REGION Network 54: Step[155] : Main P&P 1,2 Z-Axis Wait Pos
   RUNG wire#powerrail
      { S7_Templates := "SrcType := DInt" } EQ_Contact(in1 := "Unit1.Em4.ControlNodes".mainPnP.sequence.status.currentStep, in2 := #JOB_1_STEP_55)
      Contact( "Unit1.Em4.ControlNodes".mainPnP.sequence.status.seqActive )
      wire#w1
      Contact( #TRUE )
      wire#w2
      I_Contact( "Unit1.Em4.ControlNodes".cm.softCam.anodeMainPnP1AxisZ.upPos.inPos )
      wire#w3
      Coil( "Unit1.Em4.ControlNodes".mainPnP."step".action1[155] )
   END_RUNG
   RUNG wire#w2
      I_Contact( "Unit1.Em4.ControlNodes".cm.softCam.anodeMainPnP2AxisZ.upPos.inPos )
   END_RUNG wire#w3
   RUNG wire#w2
      Contact( "Unit1.Em4.ControlNodes".cm.softCam.anodeMainPnP1AxisZ.upPos.inPos )
      Contact( "Unit1.Em4.ControlNodes".cm.softCam.anodeMainPnP2AxisZ.upPos.inPos )
      Coil( "Unit1.Em4.ControlNodes".mainPnP."step".transition1[155] )
   END_RUNG
   RUNG wire#w1
      Contact( "Unit1.Em4.ControlNodes".mainPnP."step".transition1[155] )
      wire#w4
      { S7_Templates := "SrcType := DInt" } EQ_Contact(in1 := "Unit1.EmData".remainValue, in2 := 1)
      Contact( "Unit1.EmNodes".emRelations.em05.sequence.Spare1.selectJobStatus[1].completed )
      wire#w5
      Coil( "Unit1.Em4.ControlNodes".mainPnP."step".transition2[155] )
   END_RUNG
   RUNG wire#w4
      { S7_Templates := "SrcType := DInt" } EQ_Contact(in1 := "Unit1.EmData".remainValue, in2 := 0)
   END_RUNG wire#w5
   RUNG wire#w1
      Contact( "Unit1.Em4.ControlNodes".mainPnP."step".transition2[155] )
      { S7_Templates := "time_type := Time" } #statTonTime[155].TON(pt := #delayTime, et =>)
      Move(in := #JOB_1_STEP_80, out1 => "Unit1.Em4.ControlNodes".mainPnP.sequence.status.nextStep)
   END_RUNG
   // the same network as SCL:
   #_w1 := ("Unit1.Em4.ControlNodes".mainPnP.sequence.status.currentStep = #JOB_1_STEP_55) AND "Unit1.Em4.ControlNodes".mainPnP.sequence.status.seqActive;
   #_w2 := #_w1 AND #TRUE;
   "Unit1.Em4.ControlNodes".mainPnP."step".action1[155] := #_w2 AND (NOT "Unit1.Em4.ControlNodes".cm.softCam.anodeMainPnP1AxisZ.upPos.inPos OR NOT "Unit1.Em4.ControlNodes".cm.softCam.anodeMainPnP2AxisZ.upPos.inPos);
   "Unit1.Em4.ControlNodes".mainPnP."step".transition1[155] := #_w2 AND "Unit1.Em4.ControlNodes".cm.softCam.anodeMainPnP1AxisZ.upPos.inPos AND "Unit1.Em4.ControlNodes".cm.softCam.anodeMainPnP2AxisZ.upPos.inPos;
   "Unit1.Em4.ControlNodes".mainPnP."step".transition2[155] := #_w1 AND "Unit1.Em4.ControlNodes".mainPnP."step".transition1[155] AND ((("Unit1.EmData".remainValue = 1) AND "Unit1.EmNodes".emRelations.em05.sequence.Spare1.selectJobStatus[1].completed) OR ("Unit1.EmData".remainValue = 0));
   #statTonTime[155].TON(IN := #_w1 AND "Unit1.Em4.ControlNodes".mainPnP."step".transition2[155],
                         PT := #delayTime);
   IF #statTonTime[155].Q THEN
       "Unit1.Em4.ControlNodes".mainPnP.sequence.status.nextStep := #JOB_1_STEP_80;
   END_IF;
END_REGION

REGION Network 56: Step[180] : Main P&P 1,2 X-Axis Unload Pos
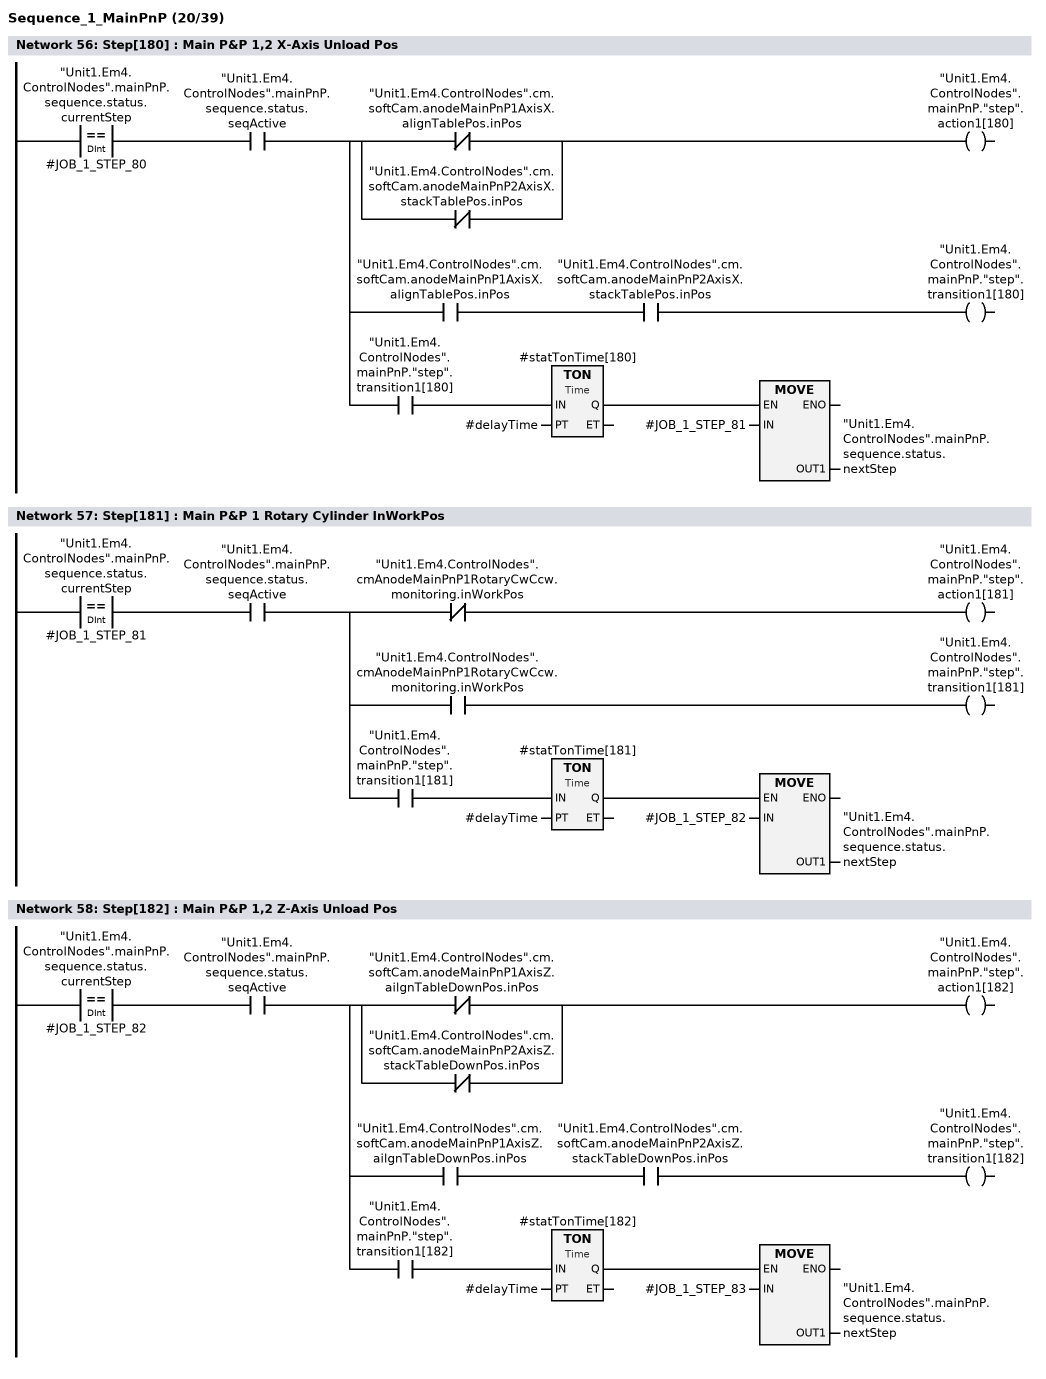
   RUNG wire#powerrail
      { S7_Templates := "SrcType := DInt" } EQ_Contact(in1 := "Unit1.Em4.ControlNodes".mainPnP.sequence.status.currentStep, in2 := #JOB_1_STEP_80)
      Contact( "Unit1.Em4.ControlNodes".mainPnP.sequence.status.seqActive )
      wire#w1
      I_Contact( "Unit1.Em4.ControlNodes".cm.softCam.anodeMainPnP1AxisX.alignTablePos.inPos )
      wire#w2
      Coil( "Unit1.Em4.ControlNodes".mainPnP."step".action1[180] )
   END_RUNG
   RUNG wire#w1
      I_Contact( "Unit1.Em4.ControlNodes".cm.softCam.anodeMainPnP2AxisX.stackTablePos.inPos )
   END_RUNG wire#w2
   RUNG wire#w1
      Contact( "Unit1.Em4.ControlNodes".cm.softCam.anodeMainPnP1AxisX.alignTablePos.inPos )
      Contact( "Unit1.Em4.ControlNodes".cm.softCam.anodeMainPnP2AxisX.stackTablePos.inPos )
      Coil( "Unit1.Em4.ControlNodes".mainPnP."step".transition1[180] )
   END_RUNG
   RUNG wire#w1
      Contact( "Unit1.Em4.ControlNodes".mainPnP."step".transition1[180] )
      { S7_Templates := "time_type := Time" } #statTonTime[180].TON(pt := #delayTime, et =>)
      Move(in := #JOB_1_STEP_81, out1 => "Unit1.Em4.ControlNodes".mainPnP.sequence.status.nextStep)
   END_RUNG
   // the same network as SCL:
   #_w1 := ("Unit1.Em4.ControlNodes".mainPnP.sequence.status.currentStep = #JOB_1_STEP_80) AND "Unit1.Em4.ControlNodes".mainPnP.sequence.status.seqActive;
   "Unit1.Em4.ControlNodes".mainPnP."step".action1[180] := #_w1 AND (NOT "Unit1.Em4.ControlNodes".cm.softCam.anodeMainPnP1AxisX.alignTablePos.inPos OR NOT "Unit1.Em4.ControlNodes".cm.softCam.anodeMainPnP2AxisX.stackTablePos.inPos);
   "Unit1.Em4.ControlNodes".mainPnP."step".transition1[180] := #_w1 AND "Unit1.Em4.ControlNodes".cm.softCam.anodeMainPnP1AxisX.alignTablePos.inPos AND "Unit1.Em4.ControlNodes".cm.softCam.anodeMainPnP2AxisX.stackTablePos.inPos;
   #statTonTime[180].TON(IN := #_w1 AND "Unit1.Em4.ControlNodes".mainPnP."step".transition1[180],
                         PT := #delayTime);
   IF #statTonTime[180].Q THEN
       "Unit1.Em4.ControlNodes".mainPnP.sequence.status.nextStep := #JOB_1_STEP_81;
   END_IF;
END_REGION

REGION Network 57: Step[181] : Main P&P 1 Rotary Cylinder InWorkPos
   RUNG wire#powerrail
      { S7_Templates := "SrcType := DInt" } EQ_Contact(in1 := "Unit1.Em4.ControlNodes".mainPnP.sequence.status.currentStep, in2 := #JOB_1_STEP_81)
      Contact( "Unit1.Em4.ControlNodes".mainPnP.sequence.status.seqActive )
      wire#w1
      I_Contact( "Unit1.Em4.ControlNodes".cmAnodeMainPnP1RotaryCwCcw.monitoring.inWorkPos )
      Coil( "Unit1.Em4.ControlNodes".mainPnP."step".action1[181] )
   END_RUNG
   RUNG wire#w1
      Contact( "Unit1.Em4.ControlNodes".cmAnodeMainPnP1RotaryCwCcw.monitoring.inWorkPos )
      Coil( "Unit1.Em4.ControlNodes".mainPnP."step".transition1[181] )
   END_RUNG
   RUNG wire#w1
      Contact( "Unit1.Em4.ControlNodes".mainPnP."step".transition1[181] )
      { S7_Templates := "time_type := Time" } #statTonTime[181].TON(pt := #delayTime, et =>)
      Move(in := #JOB_1_STEP_82, out1 => "Unit1.Em4.ControlNodes".mainPnP.sequence.status.nextStep)
   END_RUNG
   // the same network as SCL:
   #_w1 := ("Unit1.Em4.ControlNodes".mainPnP.sequence.status.currentStep = #JOB_1_STEP_81) AND "Unit1.Em4.ControlNodes".mainPnP.sequence.status.seqActive;
   "Unit1.Em4.ControlNodes".mainPnP."step".action1[181] := #_w1 AND NOT "Unit1.Em4.ControlNodes".cmAnodeMainPnP1RotaryCwCcw.monitoring.inWorkPos;
   "Unit1.Em4.ControlNodes".mainPnP."step".transition1[181] := #_w1 AND "Unit1.Em4.ControlNodes".cmAnodeMainPnP1RotaryCwCcw.monitoring.inWorkPos;
   #statTonTime[181].TON(IN := #_w1 AND "Unit1.Em4.ControlNodes".mainPnP."step".transition1[181],
                         PT := #delayTime);
   IF #statTonTime[181].Q THEN
       "Unit1.Em4.ControlNodes".mainPnP.sequence.status.nextStep := #JOB_1_STEP_82;
   END_IF;
END_REGION

REGION Network 58: Step[182] : Main P&P 1,2 Z-Axis Unload Pos
   RUNG wire#powerrail
      { S7_Templates := "SrcType := DInt" } EQ_Contact(in1 := "Unit1.Em4.ControlNodes".mainPnP.sequence.status.currentStep, in2 := #JOB_1_STEP_82)
      Contact( "Unit1.Em4.ControlNodes".mainPnP.sequence.status.seqActive )
      wire#w1
      I_Contact( "Unit1.Em4.ControlNodes".cm.softCam.anodeMainPnP1AxisZ.ailgnTableDownPos.inPos )
      wire#w2
      Coil( "Unit1.Em4.ControlNodes".mainPnP."step".action1[182] )
   END_RUNG
   RUNG wire#w1
      I_Contact( "Unit1.Em4.ControlNodes".cm.softCam.anodeMainPnP2AxisZ.stackTableDownPos.inPos )
   END_RUNG wire#w2
   RUNG wire#w1
      Contact( "Unit1.Em4.ControlNodes".cm.softCam.anodeMainPnP1AxisZ.ailgnTableDownPos.inPos )
      Contact( "Unit1.Em4.ControlNodes".cm.softCam.anodeMainPnP2AxisZ.stackTableDownPos.inPos )
      Coil( "Unit1.Em4.ControlNodes".mainPnP."step".transition1[182] )
   END_RUNG
   RUNG wire#w1
      Contact( "Unit1.Em4.ControlNodes".mainPnP."step".transition1[182] )
      { S7_Templates := "time_type := Time" } #statTonTime[182].TON(pt := #delayTime, et =>)
      Move(in := #JOB_1_STEP_83, out1 => "Unit1.Em4.ControlNodes".mainPnP.sequence.status.nextStep)
   END_RUNG
   // the same network as SCL:
   #_w1 := ("Unit1.Em4.ControlNodes".mainPnP.sequence.status.currentStep = #JOB_1_STEP_82) AND "Unit1.Em4.ControlNodes".mainPnP.sequence.status.seqActive;
   "Unit1.Em4.ControlNodes".mainPnP."step".action1[182] := #_w1 AND (NOT "Unit1.Em4.ControlNodes".cm.softCam.anodeMainPnP1AxisZ.ailgnTableDownPos.inPos OR NOT "Unit1.Em4.ControlNodes".cm.softCam.anodeMainPnP2AxisZ.stackTableDownPos.inPos);
   "Unit1.Em4.ControlNodes".mainPnP."step".transition1[182] := #_w1 AND "Unit1.Em4.ControlNodes".cm.softCam.anodeMainPnP1AxisZ.ailgnTableDownPos.inPos AND "Unit1.Em4.ControlNodes".cm.softCam.anodeMainPnP2AxisZ.stackTableDownPos.inPos;
   #statTonTime[182].TON(IN := #_w1 AND "Unit1.Em4.ControlNodes".mainPnP."step".transition1[182],
                         PT := #delayTime);
   IF #statTonTime[182].Q THEN
       "Unit1.Em4.ControlNodes".mainPnP.sequence.status.nextStep := #JOB_1_STEP_83;
   END_IF;
END_REGION

REGION Network 59: Step[183] : Main P&P → Align Table [Unloading Ready]
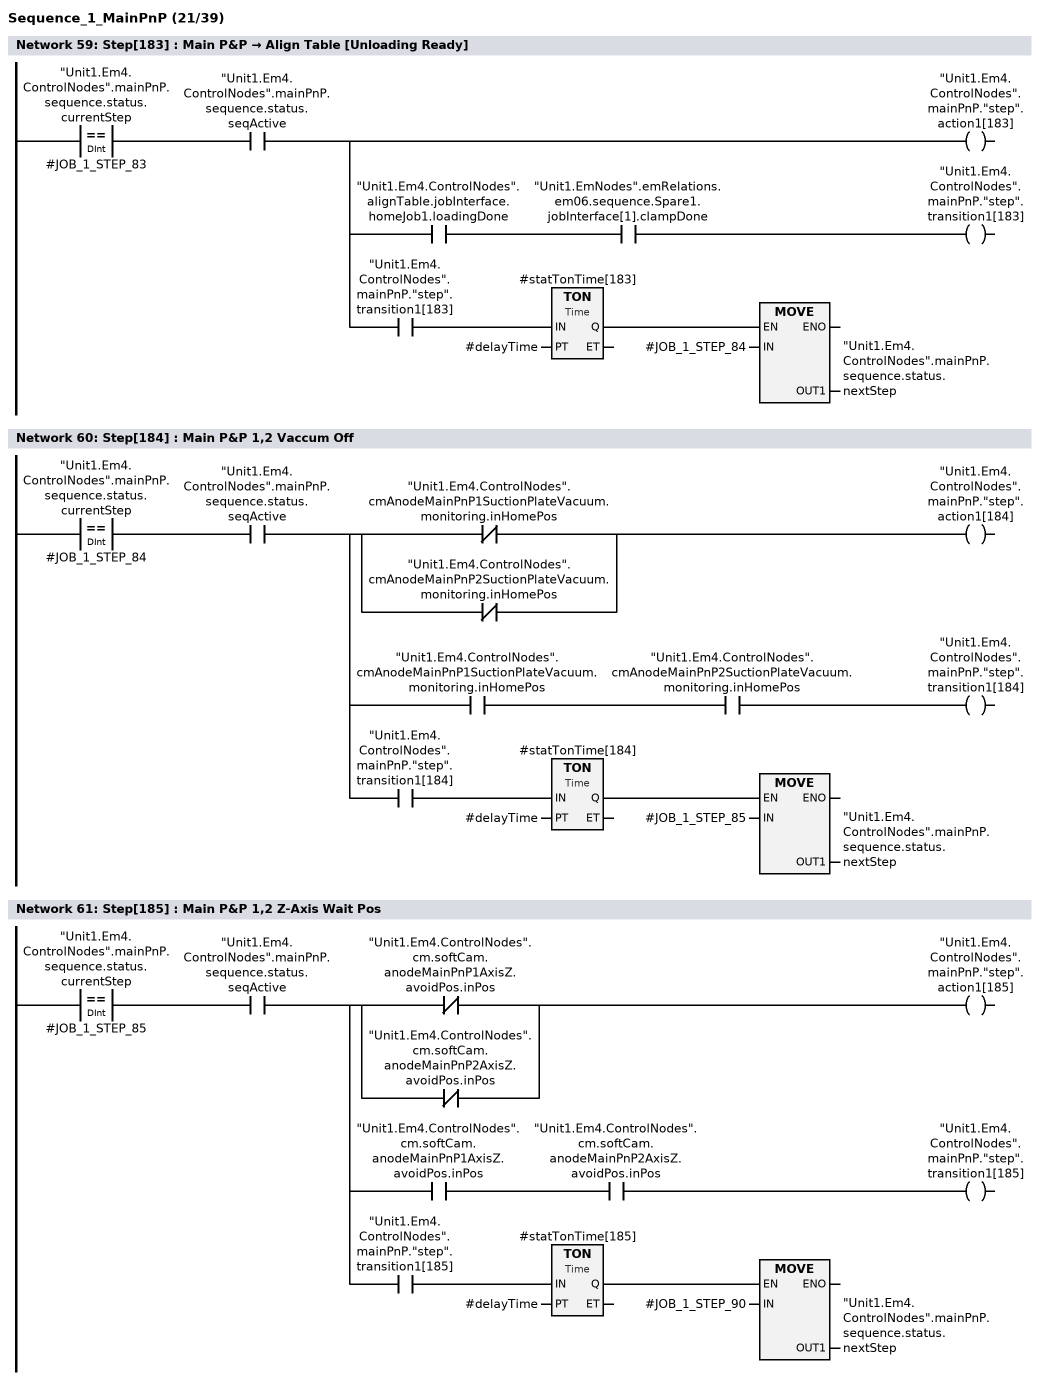
   RUNG wire#powerrail
      { S7_Templates := "SrcType := DInt" } EQ_Contact(in1 := "Unit1.Em4.ControlNodes".mainPnP.sequence.status.currentStep, in2 := #JOB_1_STEP_83)
      Contact( "Unit1.Em4.ControlNodes".mainPnP.sequence.status.seqActive )
      wire#w1
      Coil( "Unit1.Em4.ControlNodes".mainPnP."step".action1[183] )
   END_RUNG
   RUNG wire#w1
      Contact( "Unit1.Em4.ControlNodes".alignTable.jobInterface.homeJob1.loadingDone )
      Contact( "Unit1.EmNodes".emRelations.em06.sequence.Spare1.jobInterface[1].clampDone )
      Coil( "Unit1.Em4.ControlNodes".mainPnP."step".transition1[183] )
   END_RUNG
   RUNG wire#w1
      Contact( "Unit1.Em4.ControlNodes".mainPnP."step".transition1[183] )
      { S7_Templates := "time_type := Time" } #statTonTime[183].TON(pt := #delayTime, et =>)
      Move(in := #JOB_1_STEP_84, out1 => "Unit1.Em4.ControlNodes".mainPnP.sequence.status.nextStep)
   END_RUNG
   // the same network as SCL:
   "Unit1.Em4.ControlNodes".mainPnP."step".action1[183] := ("Unit1.Em4.ControlNodes".mainPnP.sequence.status.currentStep = #JOB_1_STEP_83) AND "Unit1.Em4.ControlNodes".mainPnP.sequence.status.seqActive;
   "Unit1.Em4.ControlNodes".mainPnP."step".transition1[183] := ("Unit1.Em4.ControlNodes".mainPnP.sequence.status.currentStep = #JOB_1_STEP_83) AND "Unit1.Em4.ControlNodes".mainPnP.sequence.status.seqActive AND "Unit1.Em4.ControlNodes".alignTable.jobInterface.homeJob1.loadingDone AND "Unit1.EmNodes".emRelations.em06.sequence.Spare1.jobInterface[1].clampDone;
   #statTonTime[183].TON(IN := ("Unit1.Em4.ControlNodes".mainPnP.sequence.status.currentStep = #JOB_1_STEP_83) AND "Unit1.Em4.ControlNodes".mainPnP.sequence.status.seqActive AND "Unit1.Em4.ControlNodes".mainPnP."step".transition1[183],
                         PT := #delayTime);
   IF #statTonTime[183].Q THEN
       "Unit1.Em4.ControlNodes".mainPnP.sequence.status.nextStep := #JOB_1_STEP_84;
   END_IF;
END_REGION

REGION Network 60: Step[184] : Main P&P 1,2 Vaccum Off
   RUNG wire#powerrail
      { S7_Templates := "SrcType := DInt" } EQ_Contact(in1 := "Unit1.Em4.ControlNodes".mainPnP.sequence.status.currentStep, in2 := #JOB_1_STEP_84)
      Contact( "Unit1.Em4.ControlNodes".mainPnP.sequence.status.seqActive )
      wire#w1
      I_Contact( "Unit1.Em4.ControlNodes".cmAnodeMainPnP1SuctionPlateVacuum.monitoring.inHomePos )
      wire#w2
      Coil( "Unit1.Em4.ControlNodes".mainPnP."step".action1[184] )
   END_RUNG
   RUNG wire#w1
      I_Contact( "Unit1.Em4.ControlNodes".cmAnodeMainPnP2SuctionPlateVacuum.monitoring.inHomePos )
   END_RUNG wire#w2
   RUNG wire#w1
      Contact( "Unit1.Em4.ControlNodes".cmAnodeMainPnP1SuctionPlateVacuum.monitoring.inHomePos )
      Contact( "Unit1.Em4.ControlNodes".cmAnodeMainPnP2SuctionPlateVacuum.monitoring.inHomePos )
      Coil( "Unit1.Em4.ControlNodes".mainPnP."step".transition1[184] )
   END_RUNG
   RUNG wire#w1
      Contact( "Unit1.Em4.ControlNodes".mainPnP."step".transition1[184] )
      { S7_Templates := "time_type := Time" } #statTonTime[184].TON(pt := #delayTime, et =>)
      Move(in := #JOB_1_STEP_85, out1 => "Unit1.Em4.ControlNodes".mainPnP.sequence.status.nextStep)
   END_RUNG
   // the same network as SCL:
   #_w1 := ("Unit1.Em4.ControlNodes".mainPnP.sequence.status.currentStep = #JOB_1_STEP_84) AND "Unit1.Em4.ControlNodes".mainPnP.sequence.status.seqActive;
   "Unit1.Em4.ControlNodes".mainPnP."step".action1[184] := #_w1 AND (NOT "Unit1.Em4.ControlNodes".cmAnodeMainPnP1SuctionPlateVacuum.monitoring.inHomePos OR NOT "Unit1.Em4.ControlNodes".cmAnodeMainPnP2SuctionPlateVacuum.monitoring.inHomePos);
   "Unit1.Em4.ControlNodes".mainPnP."step".transition1[184] := #_w1 AND "Unit1.Em4.ControlNodes".cmAnodeMainPnP1SuctionPlateVacuum.monitoring.inHomePos AND "Unit1.Em4.ControlNodes".cmAnodeMainPnP2SuctionPlateVacuum.monitoring.inHomePos;
   #statTonTime[184].TON(IN := #_w1 AND "Unit1.Em4.ControlNodes".mainPnP."step".transition1[184],
                         PT := #delayTime);
   IF #statTonTime[184].Q THEN
       "Unit1.Em4.ControlNodes".mainPnP.sequence.status.nextStep := #JOB_1_STEP_85;
   END_IF;
END_REGION

REGION Network 61: Step[185] : Main P&P 1,2 Z-Axis Wait Pos
   RUNG wire#powerrail
      { S7_Templates := "SrcType := DInt" } EQ_Contact(in1 := "Unit1.Em4.ControlNodes".mainPnP.sequence.status.currentStep, in2 := #JOB_1_STEP_85)
      Contact( "Unit1.Em4.ControlNodes".mainPnP.sequence.status.seqActive )
      wire#w1
      I_Contact( "Unit1.Em4.ControlNodes".cm.softCam.anodeMainPnP1AxisZ.avoidPos.inPos )
      wire#w2
      Coil( "Unit1.Em4.ControlNodes".mainPnP."step".action1[185] )
   END_RUNG
   RUNG wire#w1
      I_Contact( "Unit1.Em4.ControlNodes".cm.softCam.anodeMainPnP2AxisZ.avoidPos.inPos )
   END_RUNG wire#w2
   RUNG wire#w1
      Contact( "Unit1.Em4.ControlNodes".cm.softCam.anodeMainPnP1AxisZ.avoidPos.inPos )
      Contact( "Unit1.Em4.ControlNodes".cm.softCam.anodeMainPnP2AxisZ.avoidPos.inPos )
      Coil( "Unit1.Em4.ControlNodes".mainPnP."step".transition1[185] )
   END_RUNG
   RUNG wire#w1
      Contact( "Unit1.Em4.ControlNodes".mainPnP."step".transition1[185] )
      { S7_Templates := "time_type := Time" } #statTonTime[185].TON(pt := #delayTime, et =>)
      Move(in := #JOB_1_STEP_90, out1 => "Unit1.Em4.ControlNodes".mainPnP.sequence.status.nextStep)
   END_RUNG
   // the same network as SCL:
   #_w1 := ("Unit1.Em4.ControlNodes".mainPnP.sequence.status.currentStep = #JOB_1_STEP_85) AND "Unit1.Em4.ControlNodes".mainPnP.sequence.status.seqActive;
   "Unit1.Em4.ControlNodes".mainPnP."step".action1[185] := #_w1 AND (NOT "Unit1.Em4.ControlNodes".cm.softCam.anodeMainPnP1AxisZ.avoidPos.inPos OR NOT "Unit1.Em4.ControlNodes".cm.softCam.anodeMainPnP2AxisZ.avoidPos.inPos);
   "Unit1.Em4.ControlNodes".mainPnP."step".transition1[185] := #_w1 AND "Unit1.Em4.ControlNodes".cm.softCam.anodeMainPnP1AxisZ.avoidPos.inPos AND "Unit1.Em4.ControlNodes".cm.softCam.anodeMainPnP2AxisZ.avoidPos.inPos;
   #statTonTime[185].TON(IN := #_w1 AND "Unit1.Em4.ControlNodes".mainPnP."step".transition1[185],
                         PT := #delayTime);
   IF #statTonTime[185].Q THEN
       "Unit1.Em4.ControlNodes".mainPnP.sequence.status.nextStep := #JOB_1_STEP_90;
   END_IF;
END_REGION

REGION Network 62: Step[190] : JOB[1] Step End
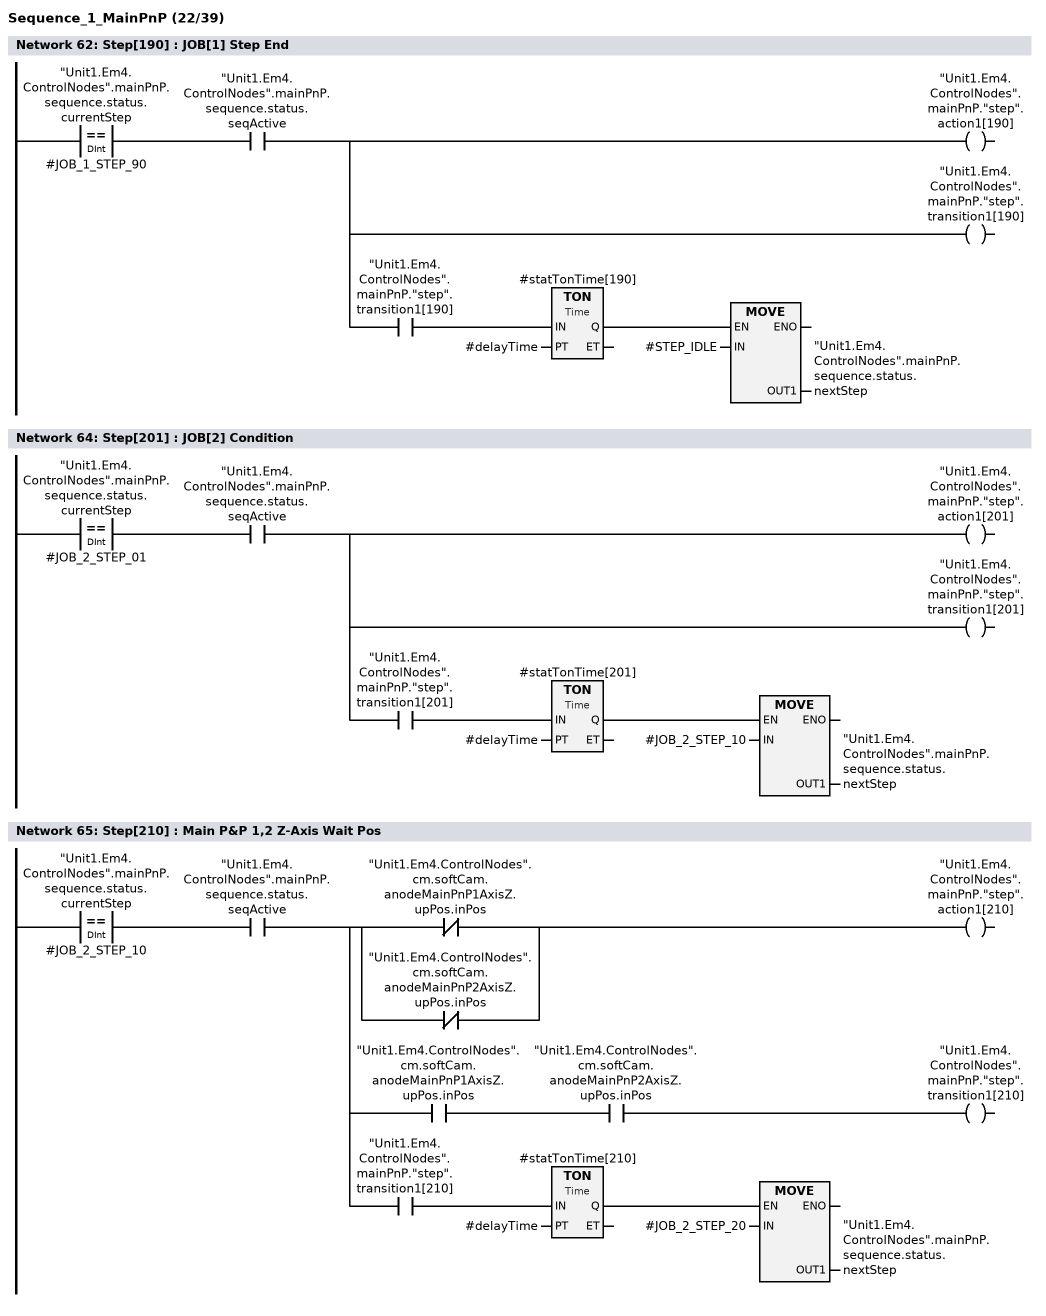
   RUNG wire#powerrail
      { S7_Templates := "SrcType := DInt" } EQ_Contact(in1 := "Unit1.Em4.ControlNodes".mainPnP.sequence.status.currentStep, in2 := #JOB_1_STEP_90)
      Contact( "Unit1.Em4.ControlNodes".mainPnP.sequence.status.seqActive )
      wire#w1
      Coil( "Unit1.Em4.ControlNodes".mainPnP."step".action1[190] )
   END_RUNG
   RUNG wire#w1
      Coil( "Unit1.Em4.ControlNodes".mainPnP."step".transition1[190] )
   END_RUNG
   RUNG wire#w1
      Contact( "Unit1.Em4.ControlNodes".mainPnP."step".transition1[190] )
      { S7_Templates := "time_type := Time" } #statTonTime[190].TON(pt := #delayTime, et =>)
      Move(in := #STEP_IDLE, out1 => "Unit1.Em4.ControlNodes".mainPnP.sequence.status.nextStep)
   END_RUNG
   // the same network as SCL:
   "Unit1.Em4.ControlNodes".mainPnP."step".action1[190] := ("Unit1.Em4.ControlNodes".mainPnP.sequence.status.currentStep = #JOB_1_STEP_90) AND "Unit1.Em4.ControlNodes".mainPnP.sequence.status.seqActive;
   "Unit1.Em4.ControlNodes".mainPnP."step".transition1[190] := ("Unit1.Em4.ControlNodes".mainPnP.sequence.status.currentStep = #JOB_1_STEP_90) AND "Unit1.Em4.ControlNodes".mainPnP.sequence.status.seqActive;
   #statTonTime[190].TON(IN := ("Unit1.Em4.ControlNodes".mainPnP.sequence.status.currentStep = #JOB_1_STEP_90) AND "Unit1.Em4.ControlNodes".mainPnP.sequence.status.seqActive AND "Unit1.Em4.ControlNodes".mainPnP."step".transition1[190],
                         PT := #delayTime);
   IF #statTonTime[190].Q THEN
       "Unit1.Em4.ControlNodes".mainPnP.sequence.status.nextStep := #STEP_IDLE;
   END_IF;
END_REGION

REGION Network 63: *************** JOB[2] Loading ************************
END_REGION

REGION Network 64: Step[201] : JOB[2] Condition
   RUNG wire#powerrail
      { S7_Templates := "SrcType := DInt" } EQ_Contact(in1 := "Unit1.Em4.ControlNodes".mainPnP.sequence.status.currentStep, in2 := #JOB_2_STEP_01)
      Contact( "Unit1.Em4.ControlNodes".mainPnP.sequence.status.seqActive )
      wire#w1
      Coil( "Unit1.Em4.ControlNodes".mainPnP."step".action1[201] )
   END_RUNG
   RUNG wire#w1
      Coil( "Unit1.Em4.ControlNodes".mainPnP."step".transition1[201] )
   END_RUNG
   RUNG wire#w1
      Contact( "Unit1.Em4.ControlNodes".mainPnP."step".transition1[201] )
      { S7_Templates := "time_type := Time" } #statTonTime[201].TON(pt := #delayTime, et =>)
      Move(in := #JOB_2_STEP_10, out1 => "Unit1.Em4.ControlNodes".mainPnP.sequence.status.nextStep)
   END_RUNG
   // the same network as SCL:
   "Unit1.Em4.ControlNodes".mainPnP."step".action1[201] := ("Unit1.Em4.ControlNodes".mainPnP.sequence.status.currentStep = #JOB_2_STEP_01) AND "Unit1.Em4.ControlNodes".mainPnP.sequence.status.seqActive;
   "Unit1.Em4.ControlNodes".mainPnP."step".transition1[201] := ("Unit1.Em4.ControlNodes".mainPnP.sequence.status.currentStep = #JOB_2_STEP_01) AND "Unit1.Em4.ControlNodes".mainPnP.sequence.status.seqActive;
   #statTonTime[201].TON(IN := ("Unit1.Em4.ControlNodes".mainPnP.sequence.status.currentStep = #JOB_2_STEP_01) AND "Unit1.Em4.ControlNodes".mainPnP.sequence.status.seqActive AND "Unit1.Em4.ControlNodes".mainPnP."step".transition1[201],
                         PT := #delayTime);
   IF #statTonTime[201].Q THEN
       "Unit1.Em4.ControlNodes".mainPnP.sequence.status.nextStep := #JOB_2_STEP_10;
   END_IF;
END_REGION

REGION Network 65: Step[210] : Main P&P 1,2 Z-Axis Wait Pos
   RUNG wire#powerrail
      { S7_Templates := "SrcType := DInt" } EQ_Contact(in1 := "Unit1.Em4.ControlNodes".mainPnP.sequence.status.currentStep, in2 := #JOB_2_STEP_10)
      Contact( "Unit1.Em4.ControlNodes".mainPnP.sequence.status.seqActive )
      wire#w1
      I_Contact( "Unit1.Em4.ControlNodes".cm.softCam.anodeMainPnP1AxisZ.upPos.inPos )
      wire#w2
      Coil( "Unit1.Em4.ControlNodes".mainPnP."step".action1[210] )
   END_RUNG
   RUNG wire#w1
      I_Contact( "Unit1.Em4.ControlNodes".cm.softCam.anodeMainPnP2AxisZ.upPos.inPos )
   END_RUNG wire#w2
   RUNG wire#w1
      Contact( "Unit1.Em4.ControlNodes".cm.softCam.anodeMainPnP1AxisZ.upPos.inPos )
      Contact( "Unit1.Em4.ControlNodes".cm.softCam.anodeMainPnP2AxisZ.upPos.inPos )
      Coil( "Unit1.Em4.ControlNodes".mainPnP."step".transition1[210] )
   END_RUNG
   RUNG wire#w1
      Contact( "Unit1.Em4.ControlNodes".mainPnP."step".transition1[210] )
      { S7_Templates := "time_type := Time" } #statTonTime[210].TON(pt := #delayTime, et =>)
      Move(in := #JOB_2_STEP_20, out1 => "Unit1.Em4.ControlNodes".mainPnP.sequence.status.nextStep)
   END_RUNG
   // the same network as SCL:
   #_w1 := ("Unit1.Em4.ControlNodes".mainPnP.sequence.status.currentStep = #JOB_2_STEP_10) AND "Unit1.Em4.ControlNodes".mainPnP.sequence.status.seqActive;
   "Unit1.Em4.ControlNodes".mainPnP."step".action1[210] := #_w1 AND (NOT "Unit1.Em4.ControlNodes".cm.softCam.anodeMainPnP1AxisZ.upPos.inPos OR NOT "Unit1.Em4.ControlNodes".cm.softCam.anodeMainPnP2AxisZ.upPos.inPos);
   "Unit1.Em4.ControlNodes".mainPnP."step".transition1[210] := #_w1 AND "Unit1.Em4.ControlNodes".cm.softCam.anodeMainPnP1AxisZ.upPos.inPos AND "Unit1.Em4.ControlNodes".cm.softCam.anodeMainPnP2AxisZ.upPos.inPos;
   #statTonTime[210].TON(IN := #_w1 AND "Unit1.Em4.ControlNodes".mainPnP."step".transition1[210],
                         PT := #delayTime);
   IF #statTonTime[210].Q THEN
       "Unit1.Em4.ControlNodes".mainPnP.sequence.status.nextStep := #JOB_2_STEP_20;
   END_IF;
END_REGION

REGION Network 66: Step[220] : Main P&P 1,2 X-Axis Load Pos
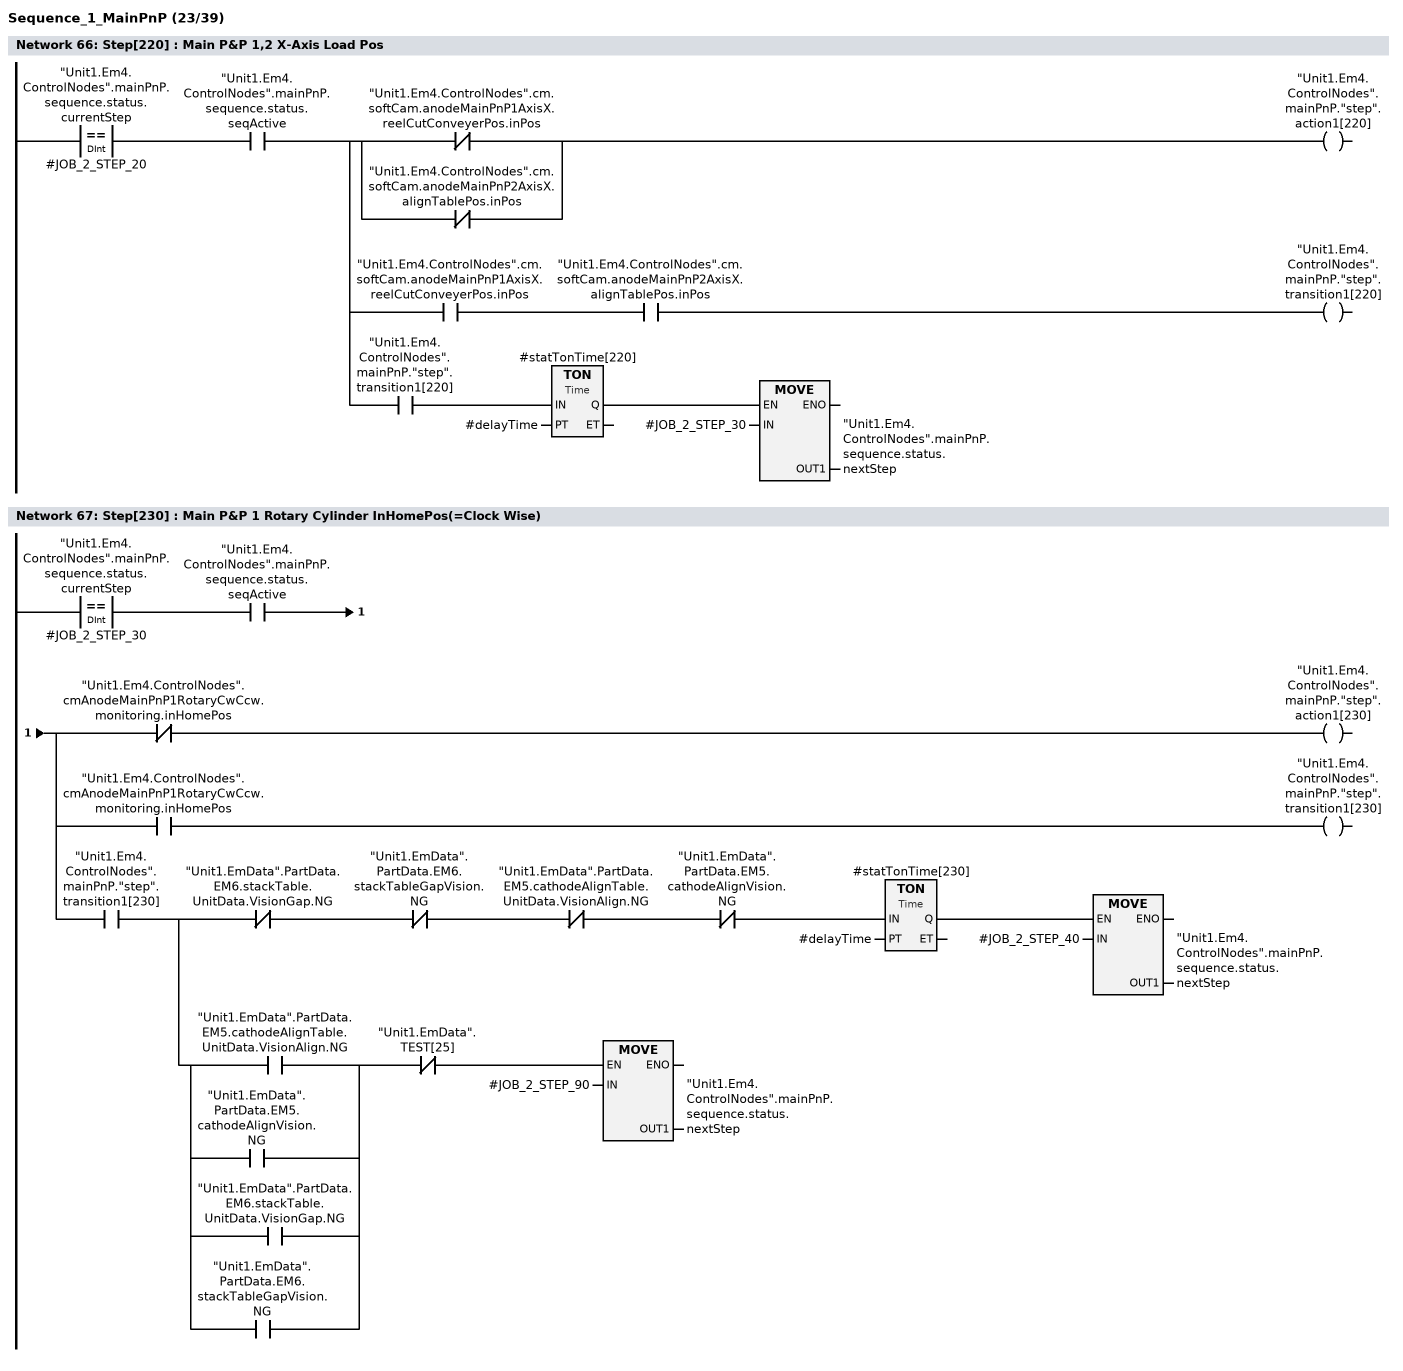
   RUNG wire#powerrail
      { S7_Templates := "SrcType := DInt" } EQ_Contact(in1 := "Unit1.Em4.ControlNodes".mainPnP.sequence.status.currentStep, in2 := #JOB_2_STEP_20)
      Contact( "Unit1.Em4.ControlNodes".mainPnP.sequence.status.seqActive )
      wire#w1
      I_Contact( "Unit1.Em4.ControlNodes".cm.softCam.anodeMainPnP1AxisX.reelCutConveyerPos.inPos )
      wire#w2
      Coil( "Unit1.Em4.ControlNodes".mainPnP."step".action1[220] )
   END_RUNG
   RUNG wire#w1
      I_Contact( "Unit1.Em4.ControlNodes".cm.softCam.anodeMainPnP2AxisX.alignTablePos.inPos )
   END_RUNG wire#w2
   RUNG wire#w1
      Contact( "Unit1.Em4.ControlNodes".cm.softCam.anodeMainPnP1AxisX.reelCutConveyerPos.inPos )
      Contact( "Unit1.Em4.ControlNodes".cm.softCam.anodeMainPnP2AxisX.alignTablePos.inPos )
      Coil( "Unit1.Em4.ControlNodes".mainPnP."step".transition1[220] )
   END_RUNG
   RUNG wire#w1
      Contact( "Unit1.Em4.ControlNodes".mainPnP."step".transition1[220] )
      { S7_Templates := "time_type := Time" } #statTonTime[220].TON(pt := #delayTime, et =>)
      Move(in := #JOB_2_STEP_30, out1 => "Unit1.Em4.ControlNodes".mainPnP.sequence.status.nextStep)
   END_RUNG
   // the same network as SCL:
   #_w1 := ("Unit1.Em4.ControlNodes".mainPnP.sequence.status.currentStep = #JOB_2_STEP_20) AND "Unit1.Em4.ControlNodes".mainPnP.sequence.status.seqActive;
   "Unit1.Em4.ControlNodes".mainPnP."step".action1[220] := #_w1 AND (NOT "Unit1.Em4.ControlNodes".cm.softCam.anodeMainPnP1AxisX.reelCutConveyerPos.inPos OR NOT "Unit1.Em4.ControlNodes".cm.softCam.anodeMainPnP2AxisX.alignTablePos.inPos);
   "Unit1.Em4.ControlNodes".mainPnP."step".transition1[220] := #_w1 AND "Unit1.Em4.ControlNodes".cm.softCam.anodeMainPnP1AxisX.reelCutConveyerPos.inPos AND "Unit1.Em4.ControlNodes".cm.softCam.anodeMainPnP2AxisX.alignTablePos.inPos;
   #statTonTime[220].TON(IN := #_w1 AND "Unit1.Em4.ControlNodes".mainPnP."step".transition1[220],
                         PT := #delayTime);
   IF #statTonTime[220].Q THEN
       "Unit1.Em4.ControlNodes".mainPnP.sequence.status.nextStep := #JOB_2_STEP_30;
   END_IF;
END_REGION

REGION Network 67: Step[230] : Main P&P 1 Rotary Cylinder InHomePos(=Clock Wise)
   RUNG wire#powerrail
      { S7_Templates := "SrcType := DInt" } EQ_Contact(in1 := "Unit1.Em4.ControlNodes".mainPnP.sequence.status.currentStep, in2 := #JOB_2_STEP_30)
      Contact( "Unit1.Em4.ControlNodes".mainPnP.sequence.status.seqActive )
      wire#w1
      I_Contact( "Unit1.Em4.ControlNodes".cmAnodeMainPnP1RotaryCwCcw.monitoring.inHomePos )
      Coil( "Unit1.Em4.ControlNodes".mainPnP."step".action1[230] )
   END_RUNG
   RUNG wire#w1
      Contact( "Unit1.Em4.ControlNodes".cmAnodeMainPnP1RotaryCwCcw.monitoring.inHomePos )
      Coil( "Unit1.Em4.ControlNodes".mainPnP."step".transition1[230] )
   END_RUNG
   RUNG wire#w1
      Contact( "Unit1.Em4.ControlNodes".mainPnP."step".transition1[230] )
      wire#w2
      I_Contact( "Unit1.EmData".PartData.EM6.stackTable.UnitData.VisionGap.NG )
      I_Contact( "Unit1.EmData".PartData.EM6.stackTableGapVision.NG )
      I_Contact( "Unit1.EmData".PartData.EM5.cathodeAlignTable.UnitData.VisionAlign.NG )
      I_Contact( "Unit1.EmData".PartData.EM5.cathodeAlignVision.NG )
      { S7_Templates := "time_type := Time" } #statTonTime[230].TON(pt := #delayTime, et =>)
      Move(in := #JOB_2_STEP_40, out1 => "Unit1.Em4.ControlNodes".mainPnP.sequence.status.nextStep)
   END_RUNG
   RUNG wire#w2
      Contact( "Unit1.EmData".PartData.EM5.cathodeAlignTable.UnitData.VisionAlign.NG )
      wire#w3
      I_Contact( "Unit1.EmData".TEST[25] )
      Move(in := #JOB_2_STEP_90, out1 => "Unit1.Em4.ControlNodes".mainPnP.sequence.status.nextStep)
   END_RUNG
   RUNG wire#w2
      Contact( "Unit1.EmData".PartData.EM5.cathodeAlignVision.NG )
   END_RUNG wire#w3
   RUNG wire#w2
      Contact( "Unit1.EmData".PartData.EM6.stackTable.UnitData.VisionGap.NG )
   END_RUNG wire#w3
   RUNG wire#w2
      Contact( "Unit1.EmData".PartData.EM6.stackTableGapVision.NG )
   END_RUNG wire#w3
   // the same network as SCL:
   #_w1 := ("Unit1.Em4.ControlNodes".mainPnP.sequence.status.currentStep = #JOB_2_STEP_30) AND "Unit1.Em4.ControlNodes".mainPnP.sequence.status.seqActive;
   "Unit1.Em4.ControlNodes".mainPnP."step".action1[230] := #_w1 AND NOT "Unit1.Em4.ControlNodes".cmAnodeMainPnP1RotaryCwCcw.monitoring.inHomePos;
   "Unit1.Em4.ControlNodes".mainPnP."step".transition1[230] := #_w1 AND "Unit1.Em4.ControlNodes".cmAnodeMainPnP1RotaryCwCcw.monitoring.inHomePos;
   #_w2 := #_w1 AND "Unit1.Em4.ControlNodes".mainPnP."step".transition1[230];
   #statTonTime[230].TON(IN := #_w2 AND NOT "Unit1.EmData".PartData.EM6.stackTable.UnitData.VisionGap.NG AND NOT "Unit1.EmData".PartData.EM6.stackTableGapVision.NG AND NOT "Unit1.EmData".PartData.EM5.cathodeAlignTable.UnitData.VisionAlign.NG AND NOT "Unit1.EmData".PartData.EM5.cathodeAlignVision.NG,
                         PT := #delayTime);
   IF #statTonTime[230].Q THEN
       "Unit1.Em4.ControlNodes".mainPnP.sequence.status.nextStep := #JOB_2_STEP_40;
   END_IF;
   IF #_w2 AND ("Unit1.EmData".PartData.EM5.cathodeAlignTable.UnitData.VisionAlign.NG OR "Unit1.EmData".PartData.EM5.cathodeAlignVision.NG OR "Unit1.EmData".PartData.EM6.stackTable.UnitData.VisionGap.NG OR "Unit1.EmData".PartData.EM6.stackTableGapVision.NG) AND NOT "Unit1.EmData".TEST[25] THEN
       "Unit1.Em4.ControlNodes".mainPnP.sequence.status.nextStep := #JOB_2_STEP_90;
   END_IF;
END_REGION

REGION Network 68: Step[240] : Main P&P 1.2 Z-Axis Load Pos
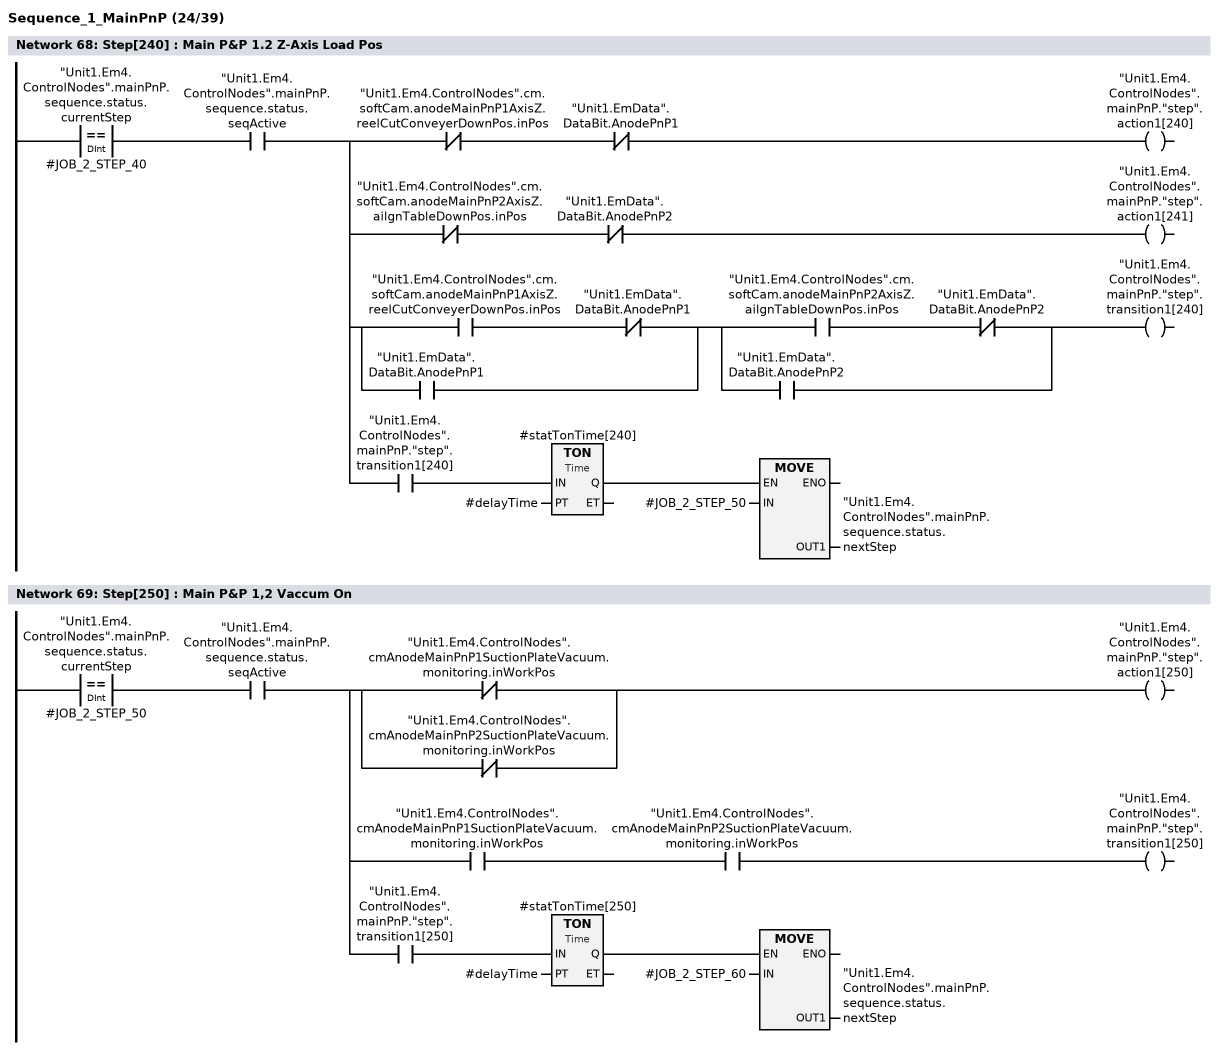
   RUNG wire#powerrail
      { S7_Templates := "SrcType := DInt" } EQ_Contact(in1 := "Unit1.Em4.ControlNodes".mainPnP.sequence.status.currentStep, in2 := #JOB_2_STEP_40)
      Contact( "Unit1.Em4.ControlNodes".mainPnP.sequence.status.seqActive )
      wire#w1
      I_Contact( "Unit1.Em4.ControlNodes".cm.softCam.anodeMainPnP1AxisZ.reelCutConveyerDownPos.inPos )
      I_Contact( "Unit1.EmData".DataBit.AnodePnP1 )
      Coil( "Unit1.Em4.ControlNodes".mainPnP."step".action1[240] )
   END_RUNG
   RUNG wire#w1
      I_Contact( "Unit1.Em4.ControlNodes".cm.softCam.anodeMainPnP2AxisZ.ailgnTableDownPos.inPos )
      I_Contact( "Unit1.EmData".DataBit.AnodePnP2 )
      Coil( "Unit1.Em4.ControlNodes".mainPnP."step".action1[241] )
   END_RUNG
   RUNG wire#w1
      Contact( "Unit1.Em4.ControlNodes".cm.softCam.anodeMainPnP1AxisZ.reelCutConveyerDownPos.inPos )
      I_Contact( "Unit1.EmData".DataBit.AnodePnP1 )
      wire#w2
      Contact( "Unit1.Em4.ControlNodes".cm.softCam.anodeMainPnP2AxisZ.ailgnTableDownPos.inPos )
      I_Contact( "Unit1.EmData".DataBit.AnodePnP2 )
      wire#w3
      Coil( "Unit1.Em4.ControlNodes".mainPnP."step".transition1[240] )
   END_RUNG
   RUNG wire#w1
      Contact( "Unit1.EmData".DataBit.AnodePnP1 )
   END_RUNG wire#w2
   RUNG wire#w2
      Contact( "Unit1.EmData".DataBit.AnodePnP2 )
   END_RUNG wire#w3
   RUNG wire#w1
      Contact( "Unit1.Em4.ControlNodes".mainPnP."step".transition1[240] )
      { S7_Templates := "time_type := Time" } #statTonTime[240].TON(pt := #delayTime, et =>)
      Move(in := #JOB_2_STEP_50, out1 => "Unit1.Em4.ControlNodes".mainPnP.sequence.status.nextStep)
   END_RUNG
   // the same network as SCL:
   #_w1 := ("Unit1.Em4.ControlNodes".mainPnP.sequence.status.currentStep = #JOB_2_STEP_40) AND "Unit1.Em4.ControlNodes".mainPnP.sequence.status.seqActive;
   "Unit1.Em4.ControlNodes".mainPnP."step".action1[240] := #_w1 AND NOT "Unit1.Em4.ControlNodes".cm.softCam.anodeMainPnP1AxisZ.reelCutConveyerDownPos.inPos AND NOT "Unit1.EmData".DataBit.AnodePnP1;
   "Unit1.Em4.ControlNodes".mainPnP."step".action1[241] := #_w1 AND NOT "Unit1.Em4.ControlNodes".cm.softCam.anodeMainPnP2AxisZ.ailgnTableDownPos.inPos AND NOT "Unit1.EmData".DataBit.AnodePnP2;
   "Unit1.Em4.ControlNodes".mainPnP."step".transition1[240] := #_w1 AND (("Unit1.Em4.ControlNodes".cm.softCam.anodeMainPnP1AxisZ.reelCutConveyerDownPos.inPos AND NOT "Unit1.EmData".DataBit.AnodePnP1) OR "Unit1.EmData".DataBit.AnodePnP1) AND (("Unit1.Em4.ControlNodes".cm.softCam.anodeMainPnP2AxisZ.ailgnTableDownPos.inPos AND NOT "Unit1.EmData".DataBit.AnodePnP2) OR "Unit1.EmData".DataBit.AnodePnP2);
   #statTonTime[240].TON(IN := #_w1 AND "Unit1.Em4.ControlNodes".mainPnP."step".transition1[240],
                         PT := #delayTime);
   IF #statTonTime[240].Q THEN
       "Unit1.Em4.ControlNodes".mainPnP.sequence.status.nextStep := #JOB_2_STEP_50;
   END_IF;
END_REGION

REGION Network 69: Step[250] : Main P&P 1,2 Vaccum On
   RUNG wire#powerrail
      { S7_Templates := "SrcType := DInt" } EQ_Contact(in1 := "Unit1.Em4.ControlNodes".mainPnP.sequence.status.currentStep, in2 := #JOB_2_STEP_50)
      Contact( "Unit1.Em4.ControlNodes".mainPnP.sequence.status.seqActive )
      wire#w1
      I_Contact( "Unit1.Em4.ControlNodes".cmAnodeMainPnP1SuctionPlateVacuum.monitoring.inWorkPos )
      wire#w2
      Coil( "Unit1.Em4.ControlNodes".mainPnP."step".action1[250] )
   END_RUNG
   RUNG wire#w1
      I_Contact( "Unit1.Em4.ControlNodes".cmAnodeMainPnP2SuctionPlateVacuum.monitoring.inWorkPos )
   END_RUNG wire#w2
   RUNG wire#w1
      Contact( "Unit1.Em4.ControlNodes".cmAnodeMainPnP1SuctionPlateVacuum.monitoring.inWorkPos )
      Contact( "Unit1.Em4.ControlNodes".cmAnodeMainPnP2SuctionPlateVacuum.monitoring.inWorkPos )
      Coil( "Unit1.Em4.ControlNodes".mainPnP."step".transition1[250] )
   END_RUNG
   RUNG wire#w1
      Contact( "Unit1.Em4.ControlNodes".mainPnP."step".transition1[250] )
      { S7_Templates := "time_type := Time" } #statTonTime[250].TON(pt := #delayTime, et =>)
      Move(in := #JOB_2_STEP_60, out1 => "Unit1.Em4.ControlNodes".mainPnP.sequence.status.nextStep)
   END_RUNG
   // the same network as SCL:
   #_w1 := ("Unit1.Em4.ControlNodes".mainPnP.sequence.status.currentStep = #JOB_2_STEP_50) AND "Unit1.Em4.ControlNodes".mainPnP.sequence.status.seqActive;
   "Unit1.Em4.ControlNodes".mainPnP."step".action1[250] := #_w1 AND (NOT "Unit1.Em4.ControlNodes".cmAnodeMainPnP1SuctionPlateVacuum.monitoring.inWorkPos OR NOT "Unit1.Em4.ControlNodes".cmAnodeMainPnP2SuctionPlateVacuum.monitoring.inWorkPos);
   "Unit1.Em4.ControlNodes".mainPnP."step".transition1[250] := #_w1 AND "Unit1.Em4.ControlNodes".cmAnodeMainPnP1SuctionPlateVacuum.monitoring.inWorkPos AND "Unit1.Em4.ControlNodes".cmAnodeMainPnP2SuctionPlateVacuum.monitoring.inWorkPos;
   #statTonTime[250].TON(IN := #_w1 AND "Unit1.Em4.ControlNodes".mainPnP."step".transition1[250],
                         PT := #delayTime);
   IF #statTonTime[250].Q THEN
       "Unit1.Em4.ControlNodes".mainPnP.sequence.status.nextStep := #JOB_2_STEP_60;
   END_IF;
END_REGION

REGION Network 70: Step[260] : Main P&P → Align Table [Loading Ready]
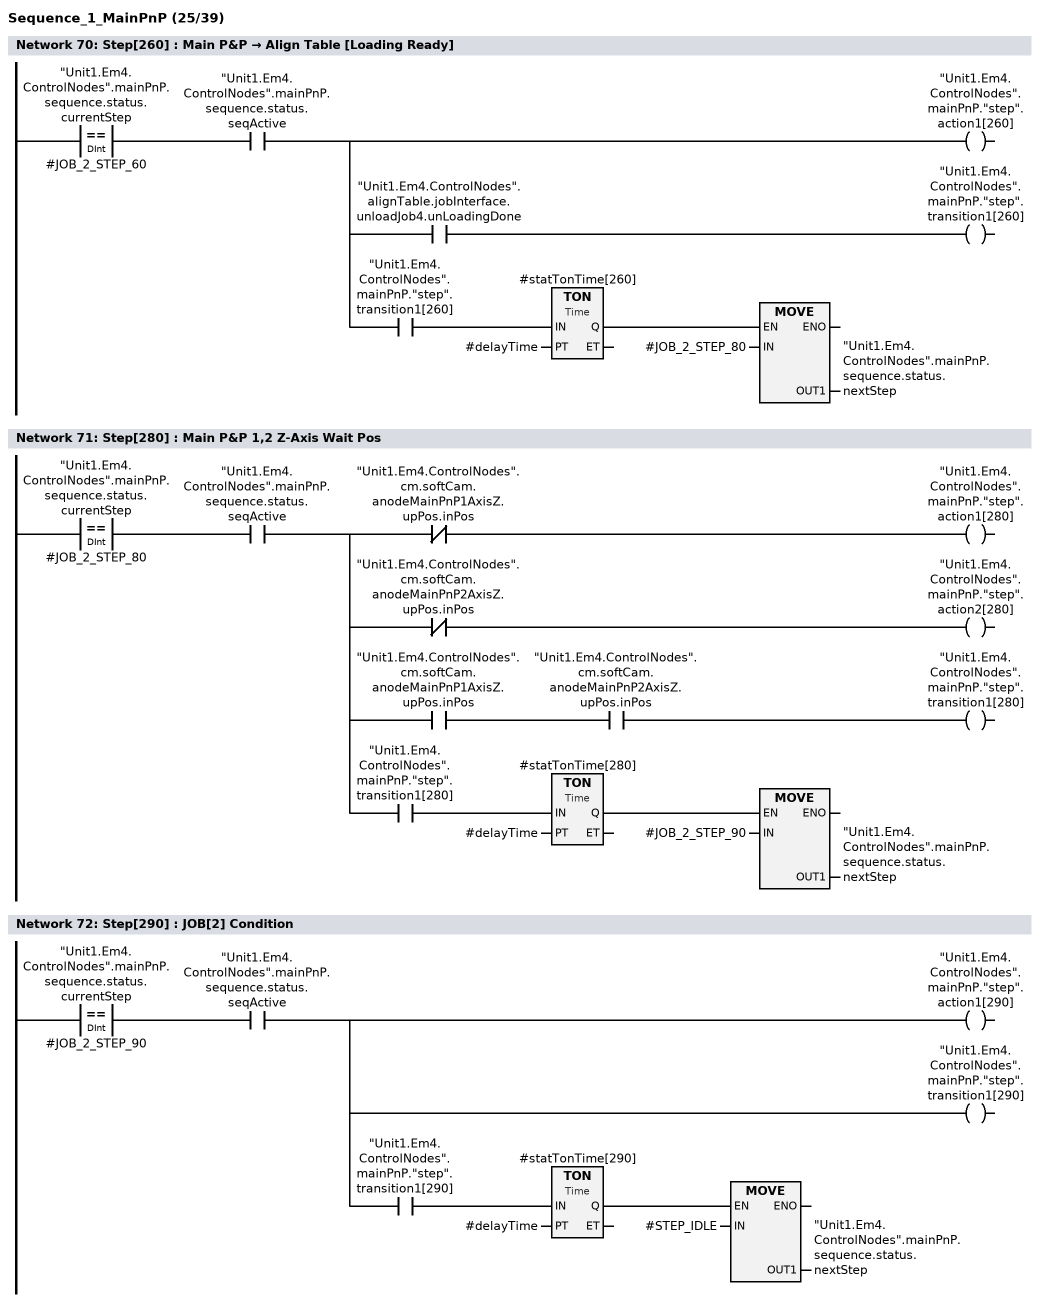
   RUNG wire#powerrail
      { S7_Templates := "SrcType := DInt" } EQ_Contact(in1 := "Unit1.Em4.ControlNodes".mainPnP.sequence.status.currentStep, in2 := #JOB_2_STEP_60)
      Contact( "Unit1.Em4.ControlNodes".mainPnP.sequence.status.seqActive )
      wire#w1
      Coil( "Unit1.Em4.ControlNodes".mainPnP."step".action1[260] )
   END_RUNG
   RUNG wire#w1
      Contact( "Unit1.Em4.ControlNodes".alignTable.jobInterface.unloadJob4.unLoadingDone )
      Coil( "Unit1.Em4.ControlNodes".mainPnP."step".transition1[260] )
   END_RUNG
   RUNG wire#w1
      Contact( "Unit1.Em4.ControlNodes".mainPnP."step".transition1[260] )
      { S7_Templates := "time_type := Time" } #statTonTime[260].TON(pt := #delayTime, et =>)
      Move(in := #JOB_2_STEP_80, out1 => "Unit1.Em4.ControlNodes".mainPnP.sequence.status.nextStep)
   END_RUNG
   // the same network as SCL:
   "Unit1.Em4.ControlNodes".mainPnP."step".action1[260] := ("Unit1.Em4.ControlNodes".mainPnP.sequence.status.currentStep = #JOB_2_STEP_60) AND "Unit1.Em4.ControlNodes".mainPnP.sequence.status.seqActive;
   "Unit1.Em4.ControlNodes".mainPnP."step".transition1[260] := ("Unit1.Em4.ControlNodes".mainPnP.sequence.status.currentStep = #JOB_2_STEP_60) AND "Unit1.Em4.ControlNodes".mainPnP.sequence.status.seqActive AND "Unit1.Em4.ControlNodes".alignTable.jobInterface.unloadJob4.unLoadingDone;
   #statTonTime[260].TON(IN := ("Unit1.Em4.ControlNodes".mainPnP.sequence.status.currentStep = #JOB_2_STEP_60) AND "Unit1.Em4.ControlNodes".mainPnP.sequence.status.seqActive AND "Unit1.Em4.ControlNodes".mainPnP."step".transition1[260],
                         PT := #delayTime);
   IF #statTonTime[260].Q THEN
       "Unit1.Em4.ControlNodes".mainPnP.sequence.status.nextStep := #JOB_2_STEP_80;
   END_IF;
END_REGION

REGION Network 71: Step[280] : Main P&P 1,2 Z-Axis Wait Pos
   RUNG wire#powerrail
      { S7_Templates := "SrcType := DInt" } EQ_Contact(in1 := "Unit1.Em4.ControlNodes".mainPnP.sequence.status.currentStep, in2 := #JOB_2_STEP_80)
      Contact( "Unit1.Em4.ControlNodes".mainPnP.sequence.status.seqActive )
      wire#w1
      I_Contact( "Unit1.Em4.ControlNodes".cm.softCam.anodeMainPnP1AxisZ.upPos.inPos )
      Coil( "Unit1.Em4.ControlNodes".mainPnP."step".action1[280] )
   END_RUNG
   RUNG wire#w1
      I_Contact( "Unit1.Em4.ControlNodes".cm.softCam.anodeMainPnP2AxisZ.upPos.inPos )
      Coil( "Unit1.Em4.ControlNodes".mainPnP."step".action2[280] )
   END_RUNG
   RUNG wire#w1
      Contact( "Unit1.Em4.ControlNodes".cm.softCam.anodeMainPnP1AxisZ.upPos.inPos )
      Contact( "Unit1.Em4.ControlNodes".cm.softCam.anodeMainPnP2AxisZ.upPos.inPos )
      Coil( "Unit1.Em4.ControlNodes".mainPnP."step".transition1[280] )
   END_RUNG
   RUNG wire#w1
      Contact( "Unit1.Em4.ControlNodes".mainPnP."step".transition1[280] )
      { S7_Templates := "time_type := Time" } #statTonTime[280].TON(pt := #delayTime, et =>)
      Move(in := #JOB_2_STEP_90, out1 => "Unit1.Em4.ControlNodes".mainPnP.sequence.status.nextStep)
   END_RUNG
   // the same network as SCL:
   #_w1 := ("Unit1.Em4.ControlNodes".mainPnP.sequence.status.currentStep = #JOB_2_STEP_80) AND "Unit1.Em4.ControlNodes".mainPnP.sequence.status.seqActive;
   "Unit1.Em4.ControlNodes".mainPnP."step".action1[280] := #_w1 AND NOT "Unit1.Em4.ControlNodes".cm.softCam.anodeMainPnP1AxisZ.upPos.inPos;
   "Unit1.Em4.ControlNodes".mainPnP."step".action2[280] := #_w1 AND NOT "Unit1.Em4.ControlNodes".cm.softCam.anodeMainPnP2AxisZ.upPos.inPos;
   "Unit1.Em4.ControlNodes".mainPnP."step".transition1[280] := #_w1 AND "Unit1.Em4.ControlNodes".cm.softCam.anodeMainPnP1AxisZ.upPos.inPos AND "Unit1.Em4.ControlNodes".cm.softCam.anodeMainPnP2AxisZ.upPos.inPos;
   #statTonTime[280].TON(IN := #_w1 AND "Unit1.Em4.ControlNodes".mainPnP."step".transition1[280],
                         PT := #delayTime);
   IF #statTonTime[280].Q THEN
       "Unit1.Em4.ControlNodes".mainPnP.sequence.status.nextStep := #JOB_2_STEP_90;
   END_IF;
END_REGION

REGION Network 72: Step[290] : JOB[2] Condition
   RUNG wire#powerrail
      { S7_Templates := "SrcType := DInt" } EQ_Contact(in1 := "Unit1.Em4.ControlNodes".mainPnP.sequence.status.currentStep, in2 := #JOB_2_STEP_90)
      Contact( "Unit1.Em4.ControlNodes".mainPnP.sequence.status.seqActive )
      wire#w1
      Coil( "Unit1.Em4.ControlNodes".mainPnP."step".action1[290] )
   END_RUNG
   RUNG wire#w1
      Coil( "Unit1.Em4.ControlNodes".mainPnP."step".transition1[290] )
   END_RUNG
   RUNG wire#w1
      Contact( "Unit1.Em4.ControlNodes".mainPnP."step".transition1[290] )
      { S7_Templates := "time_type := Time" } #statTonTime[290].TON(pt := #delayTime, et =>)
      Move(in := #STEP_IDLE, out1 => "Unit1.Em4.ControlNodes".mainPnP.sequence.status.nextStep)
   END_RUNG
   // the same network as SCL:
   "Unit1.Em4.ControlNodes".mainPnP."step".action1[290] := ("Unit1.Em4.ControlNodes".mainPnP.sequence.status.currentStep = #JOB_2_STEP_90) AND "Unit1.Em4.ControlNodes".mainPnP.sequence.status.seqActive;
   "Unit1.Em4.ControlNodes".mainPnP."step".transition1[290] := ("Unit1.Em4.ControlNodes".mainPnP.sequence.status.currentStep = #JOB_2_STEP_90) AND "Unit1.Em4.ControlNodes".mainPnP.sequence.status.seqActive;
   #statTonTime[290].TON(IN := ("Unit1.Em4.ControlNodes".mainPnP.sequence.status.currentStep = #JOB_2_STEP_90) AND "Unit1.Em4.ControlNodes".mainPnP.sequence.status.seqActive AND "Unit1.Em4.ControlNodes".mainPnP."step".transition1[290],
                         PT := #delayTime);
   IF #statTonTime[290].Q THEN
       "Unit1.Em4.ControlNodes".mainPnP.sequence.status.nextStep := #STEP_IDLE;
   END_IF;
END_REGION

REGION Network 73: *************** JOB[3] Unloading ************************
END_REGION

REGION Network 74: Step[301] : JOB[3] Condition
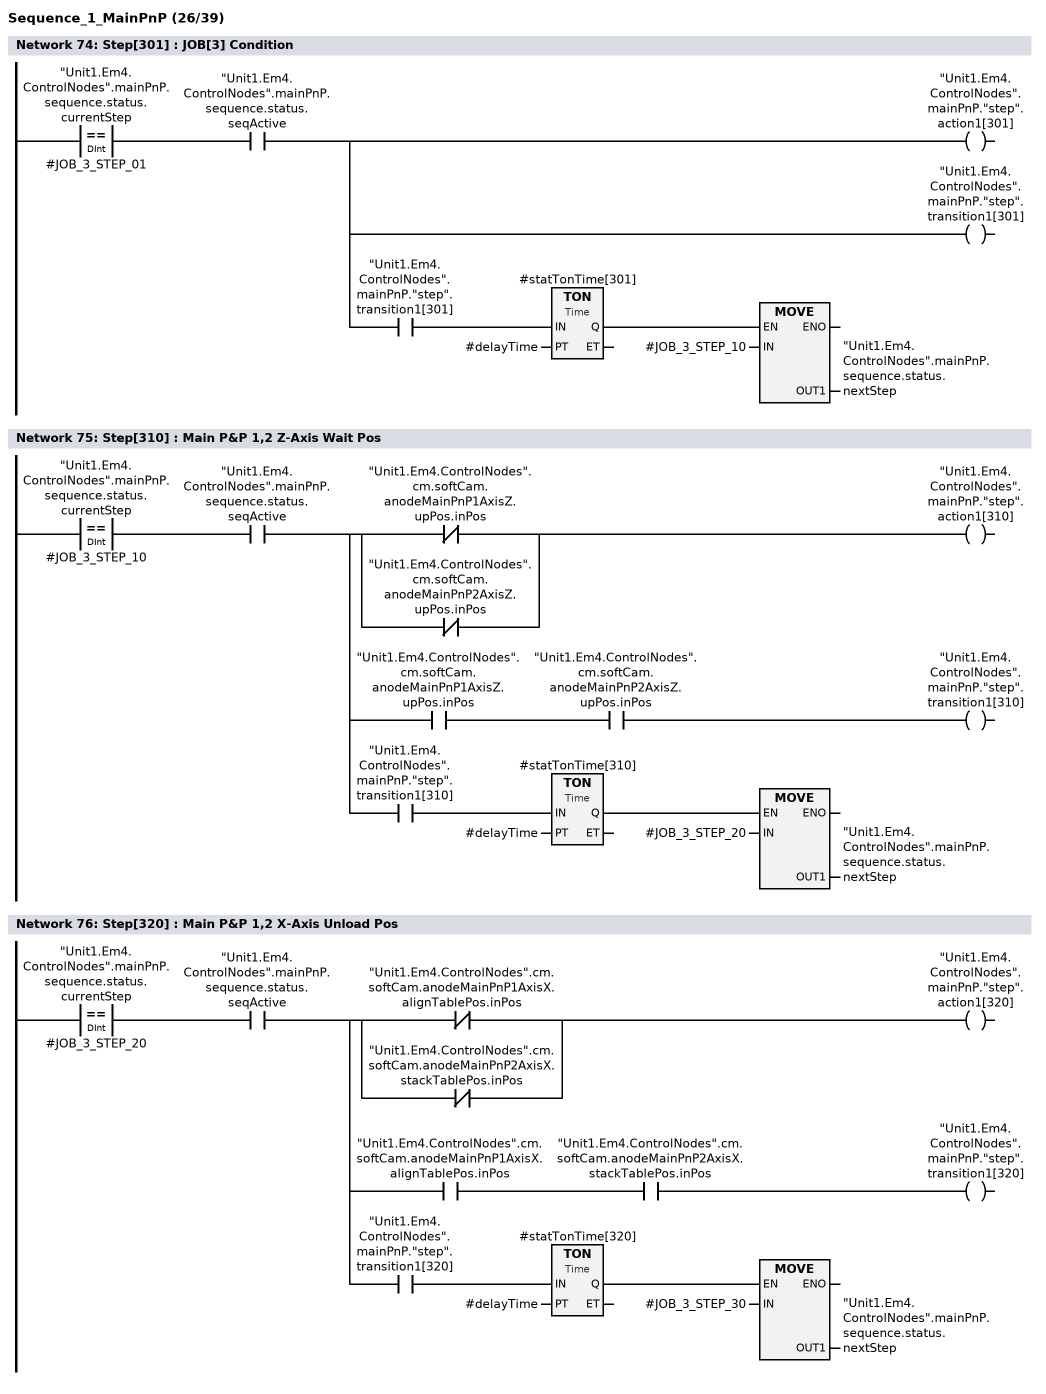
   RUNG wire#powerrail
      { S7_Templates := "SrcType := DInt" } EQ_Contact(in1 := "Unit1.Em4.ControlNodes".mainPnP.sequence.status.currentStep, in2 := #JOB_3_STEP_01)
      Contact( "Unit1.Em4.ControlNodes".mainPnP.sequence.status.seqActive )
      wire#w1
      Coil( "Unit1.Em4.ControlNodes".mainPnP."step".action1[301] )
   END_RUNG
   RUNG wire#w1
      Coil( "Unit1.Em4.ControlNodes".mainPnP."step".transition1[301] )
   END_RUNG
   RUNG wire#w1
      Contact( "Unit1.Em4.ControlNodes".mainPnP."step".transition1[301] )
      { S7_Templates := "time_type := Time" } #statTonTime[301].TON(pt := #delayTime, et =>)
      Move(in := #JOB_3_STEP_10, out1 => "Unit1.Em4.ControlNodes".mainPnP.sequence.status.nextStep)
   END_RUNG
   // the same network as SCL:
   "Unit1.Em4.ControlNodes".mainPnP."step".action1[301] := ("Unit1.Em4.ControlNodes".mainPnP.sequence.status.currentStep = #JOB_3_STEP_01) AND "Unit1.Em4.ControlNodes".mainPnP.sequence.status.seqActive;
   "Unit1.Em4.ControlNodes".mainPnP."step".transition1[301] := ("Unit1.Em4.ControlNodes".mainPnP.sequence.status.currentStep = #JOB_3_STEP_01) AND "Unit1.Em4.ControlNodes".mainPnP.sequence.status.seqActive;
   #statTonTime[301].TON(IN := ("Unit1.Em4.ControlNodes".mainPnP.sequence.status.currentStep = #JOB_3_STEP_01) AND "Unit1.Em4.ControlNodes".mainPnP.sequence.status.seqActive AND "Unit1.Em4.ControlNodes".mainPnP."step".transition1[301],
                         PT := #delayTime);
   IF #statTonTime[301].Q THEN
       "Unit1.Em4.ControlNodes".mainPnP.sequence.status.nextStep := #JOB_3_STEP_10;
   END_IF;
END_REGION

REGION Network 75: Step[310] : Main P&P 1,2 Z-Axis Wait Pos
   RUNG wire#powerrail
      { S7_Templates := "SrcType := DInt" } EQ_Contact(in1 := "Unit1.Em4.ControlNodes".mainPnP.sequence.status.currentStep, in2 := #JOB_3_STEP_10)
      Contact( "Unit1.Em4.ControlNodes".mainPnP.sequence.status.seqActive )
      wire#w1
      I_Contact( "Unit1.Em4.ControlNodes".cm.softCam.anodeMainPnP1AxisZ.upPos.inPos )
      wire#w2
      Coil( "Unit1.Em4.ControlNodes".mainPnP."step".action1[310] )
   END_RUNG
   RUNG wire#w1
      I_Contact( "Unit1.Em4.ControlNodes".cm.softCam.anodeMainPnP2AxisZ.upPos.inPos )
   END_RUNG wire#w2
   RUNG wire#w1
      Contact( "Unit1.Em4.ControlNodes".cm.softCam.anodeMainPnP1AxisZ.upPos.inPos )
      Contact( "Unit1.Em4.ControlNodes".cm.softCam.anodeMainPnP2AxisZ.upPos.inPos )
      Coil( "Unit1.Em4.ControlNodes".mainPnP."step".transition1[310] )
   END_RUNG
   RUNG wire#w1
      Contact( "Unit1.Em4.ControlNodes".mainPnP."step".transition1[310] )
      { S7_Templates := "time_type := Time" } #statTonTime[310].TON(pt := #delayTime, et =>)
      Move(in := #JOB_3_STEP_20, out1 => "Unit1.Em4.ControlNodes".mainPnP.sequence.status.nextStep)
   END_RUNG
   // the same network as SCL:
   #_w1 := ("Unit1.Em4.ControlNodes".mainPnP.sequence.status.currentStep = #JOB_3_STEP_10) AND "Unit1.Em4.ControlNodes".mainPnP.sequence.status.seqActive;
   "Unit1.Em4.ControlNodes".mainPnP."step".action1[310] := #_w1 AND (NOT "Unit1.Em4.ControlNodes".cm.softCam.anodeMainPnP1AxisZ.upPos.inPos OR NOT "Unit1.Em4.ControlNodes".cm.softCam.anodeMainPnP2AxisZ.upPos.inPos);
   "Unit1.Em4.ControlNodes".mainPnP."step".transition1[310] := #_w1 AND "Unit1.Em4.ControlNodes".cm.softCam.anodeMainPnP1AxisZ.upPos.inPos AND "Unit1.Em4.ControlNodes".cm.softCam.anodeMainPnP2AxisZ.upPos.inPos;
   #statTonTime[310].TON(IN := #_w1 AND "Unit1.Em4.ControlNodes".mainPnP."step".transition1[310],
                         PT := #delayTime);
   IF #statTonTime[310].Q THEN
       "Unit1.Em4.ControlNodes".mainPnP.sequence.status.nextStep := #JOB_3_STEP_20;
   END_IF;
END_REGION

REGION Network 76: Step[320] : Main P&P 1,2 X-Axis Unload Pos
   RUNG wire#powerrail
      { S7_Templates := "SrcType := DInt" } EQ_Contact(in1 := "Unit1.Em4.ControlNodes".mainPnP.sequence.status.currentStep, in2 := #JOB_3_STEP_20)
      Contact( "Unit1.Em4.ControlNodes".mainPnP.sequence.status.seqActive )
      wire#w1
      I_Contact( "Unit1.Em4.ControlNodes".cm.softCam.anodeMainPnP1AxisX.alignTablePos.inPos )
      wire#w2
      Coil( "Unit1.Em4.ControlNodes".mainPnP."step".action1[320] )
   END_RUNG
   RUNG wire#w1
      I_Contact( "Unit1.Em4.ControlNodes".cm.softCam.anodeMainPnP2AxisX.stackTablePos.inPos )
   END_RUNG wire#w2
   RUNG wire#w1
      Contact( "Unit1.Em4.ControlNodes".cm.softCam.anodeMainPnP1AxisX.alignTablePos.inPos )
      Contact( "Unit1.Em4.ControlNodes".cm.softCam.anodeMainPnP2AxisX.stackTablePos.inPos )
      Coil( "Unit1.Em4.ControlNodes".mainPnP."step".transition1[320] )
   END_RUNG
   RUNG wire#w1
      Contact( "Unit1.Em4.ControlNodes".mainPnP."step".transition1[320] )
      { S7_Templates := "time_type := Time" } #statTonTime[320].TON(pt := #delayTime, et =>)
      Move(in := #JOB_3_STEP_30, out1 => "Unit1.Em4.ControlNodes".mainPnP.sequence.status.nextStep)
   END_RUNG
   // the same network as SCL:
   #_w1 := ("Unit1.Em4.ControlNodes".mainPnP.sequence.status.currentStep = #JOB_3_STEP_20) AND "Unit1.Em4.ControlNodes".mainPnP.sequence.status.seqActive;
   "Unit1.Em4.ControlNodes".mainPnP."step".action1[320] := #_w1 AND (NOT "Unit1.Em4.ControlNodes".cm.softCam.anodeMainPnP1AxisX.alignTablePos.inPos OR NOT "Unit1.Em4.ControlNodes".cm.softCam.anodeMainPnP2AxisX.stackTablePos.inPos);
   "Unit1.Em4.ControlNodes".mainPnP."step".transition1[320] := #_w1 AND "Unit1.Em4.ControlNodes".cm.softCam.anodeMainPnP1AxisX.alignTablePos.inPos AND "Unit1.Em4.ControlNodes".cm.softCam.anodeMainPnP2AxisX.stackTablePos.inPos;
   #statTonTime[320].TON(IN := #_w1 AND "Unit1.Em4.ControlNodes".mainPnP."step".transition1[320],
                         PT := #delayTime);
   IF #statTonTime[320].Q THEN
       "Unit1.Em4.ControlNodes".mainPnP.sequence.status.nextStep := #JOB_3_STEP_30;
   END_IF;
END_REGION

REGION Network 77: Step[330] : Main P&P 1 Rotary Cylinder InWorkPos(=Counter Clock Wise)
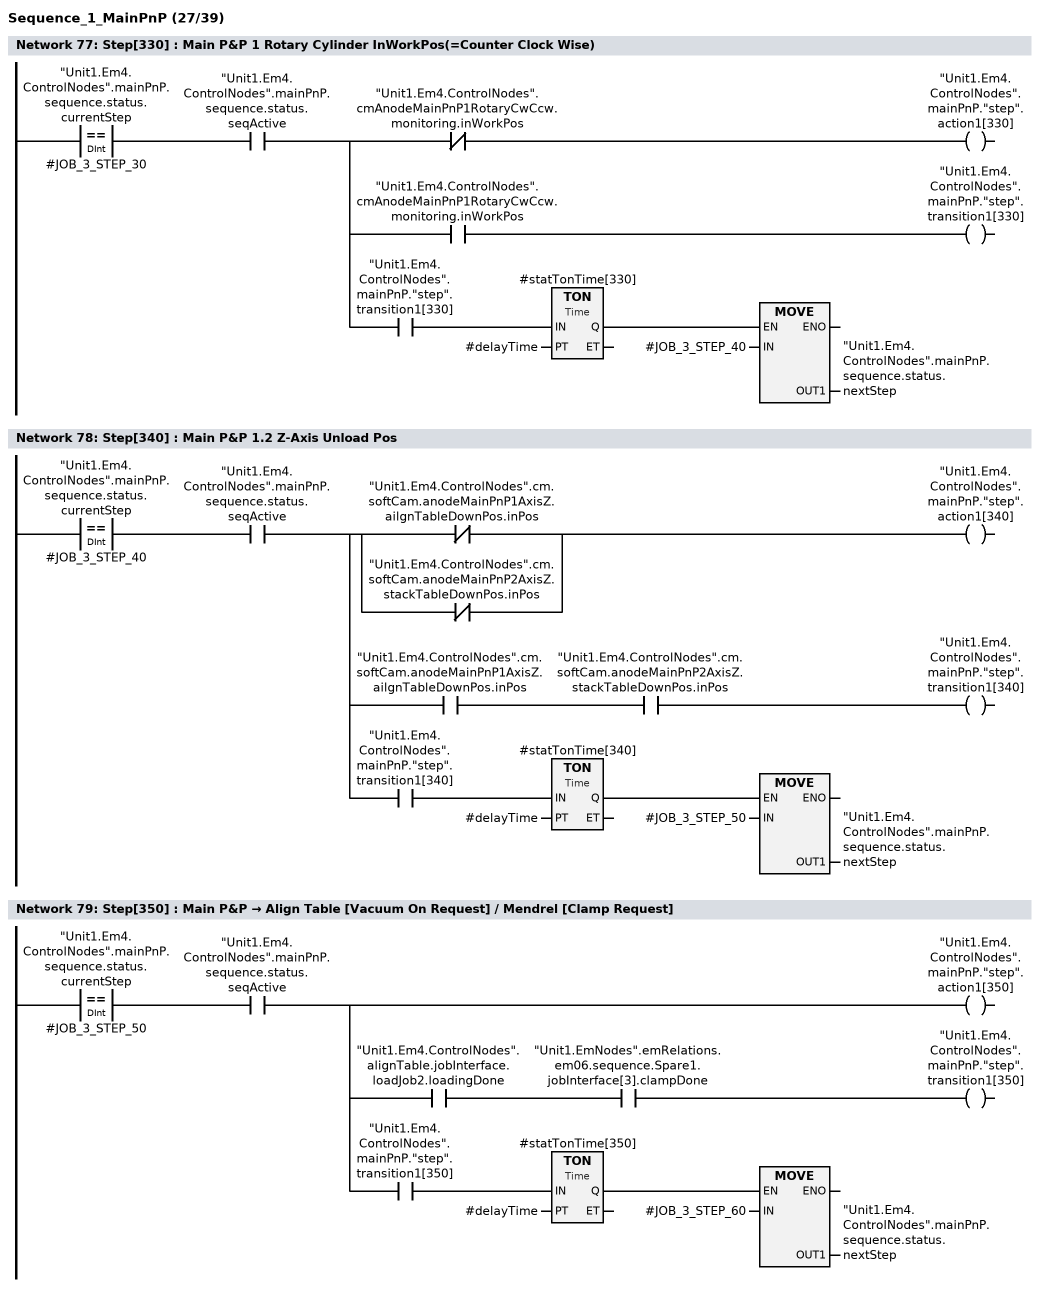
   RUNG wire#powerrail
      { S7_Templates := "SrcType := DInt" } EQ_Contact(in1 := "Unit1.Em4.ControlNodes".mainPnP.sequence.status.currentStep, in2 := #JOB_3_STEP_30)
      Contact( "Unit1.Em4.ControlNodes".mainPnP.sequence.status.seqActive )
      wire#w1
      I_Contact( "Unit1.Em4.ControlNodes".cmAnodeMainPnP1RotaryCwCcw.monitoring.inWorkPos )
      Coil( "Unit1.Em4.ControlNodes".mainPnP."step".action1[330] )
   END_RUNG
   RUNG wire#w1
      Contact( "Unit1.Em4.ControlNodes".cmAnodeMainPnP1RotaryCwCcw.monitoring.inWorkPos )
      Coil( "Unit1.Em4.ControlNodes".mainPnP."step".transition1[330] )
   END_RUNG
   RUNG wire#w1
      Contact( "Unit1.Em4.ControlNodes".mainPnP."step".transition1[330] )
      { S7_Templates := "time_type := Time" } #statTonTime[330].TON(pt := #delayTime, et =>)
      Move(in := #JOB_3_STEP_40, out1 => "Unit1.Em4.ControlNodes".mainPnP.sequence.status.nextStep)
   END_RUNG
   // the same network as SCL:
   #_w1 := ("Unit1.Em4.ControlNodes".mainPnP.sequence.status.currentStep = #JOB_3_STEP_30) AND "Unit1.Em4.ControlNodes".mainPnP.sequence.status.seqActive;
   "Unit1.Em4.ControlNodes".mainPnP."step".action1[330] := #_w1 AND NOT "Unit1.Em4.ControlNodes".cmAnodeMainPnP1RotaryCwCcw.monitoring.inWorkPos;
   "Unit1.Em4.ControlNodes".mainPnP."step".transition1[330] := #_w1 AND "Unit1.Em4.ControlNodes".cmAnodeMainPnP1RotaryCwCcw.monitoring.inWorkPos;
   #statTonTime[330].TON(IN := #_w1 AND "Unit1.Em4.ControlNodes".mainPnP."step".transition1[330],
                         PT := #delayTime);
   IF #statTonTime[330].Q THEN
       "Unit1.Em4.ControlNodes".mainPnP.sequence.status.nextStep := #JOB_3_STEP_40;
   END_IF;
END_REGION

REGION Network 78: Step[340] : Main P&P 1.2 Z-Axis Unload Pos
   RUNG wire#powerrail
      { S7_Templates := "SrcType := DInt" } EQ_Contact(in1 := "Unit1.Em4.ControlNodes".mainPnP.sequence.status.currentStep, in2 := #JOB_3_STEP_40)
      Contact( "Unit1.Em4.ControlNodes".mainPnP.sequence.status.seqActive )
      wire#w1
      I_Contact( "Unit1.Em4.ControlNodes".cm.softCam.anodeMainPnP1AxisZ.ailgnTableDownPos.inPos )
      wire#w2
      Coil( "Unit1.Em4.ControlNodes".mainPnP."step".action1[340] )
   END_RUNG
   RUNG wire#w1
      I_Contact( "Unit1.Em4.ControlNodes".cm.softCam.anodeMainPnP2AxisZ.stackTableDownPos.inPos )
   END_RUNG wire#w2
   RUNG wire#w1
      Contact( "Unit1.Em4.ControlNodes".cm.softCam.anodeMainPnP1AxisZ.ailgnTableDownPos.inPos )
      Contact( "Unit1.Em4.ControlNodes".cm.softCam.anodeMainPnP2AxisZ.stackTableDownPos.inPos )
      Coil( "Unit1.Em4.ControlNodes".mainPnP."step".transition1[340] )
   END_RUNG
   RUNG wire#w1
      Contact( "Unit1.Em4.ControlNodes".mainPnP."step".transition1[340] )
      { S7_Templates := "time_type := Time" } #statTonTime[340].TON(pt := #delayTime, et =>)
      Move(in := #JOB_3_STEP_50, out1 => "Unit1.Em4.ControlNodes".mainPnP.sequence.status.nextStep)
   END_RUNG
   // the same network as SCL:
   #_w1 := ("Unit1.Em4.ControlNodes".mainPnP.sequence.status.currentStep = #JOB_3_STEP_40) AND "Unit1.Em4.ControlNodes".mainPnP.sequence.status.seqActive;
   "Unit1.Em4.ControlNodes".mainPnP."step".action1[340] := #_w1 AND (NOT "Unit1.Em4.ControlNodes".cm.softCam.anodeMainPnP1AxisZ.ailgnTableDownPos.inPos OR NOT "Unit1.Em4.ControlNodes".cm.softCam.anodeMainPnP2AxisZ.stackTableDownPos.inPos);
   "Unit1.Em4.ControlNodes".mainPnP."step".transition1[340] := #_w1 AND "Unit1.Em4.ControlNodes".cm.softCam.anodeMainPnP1AxisZ.ailgnTableDownPos.inPos AND "Unit1.Em4.ControlNodes".cm.softCam.anodeMainPnP2AxisZ.stackTableDownPos.inPos;
   #statTonTime[340].TON(IN := #_w1 AND "Unit1.Em4.ControlNodes".mainPnP."step".transition1[340],
                         PT := #delayTime);
   IF #statTonTime[340].Q THEN
       "Unit1.Em4.ControlNodes".mainPnP.sequence.status.nextStep := #JOB_3_STEP_50;
   END_IF;
END_REGION

REGION Network 79: Step[350] : Main P&P → Align Table [Vacuum On Request] / Mendrel [Clamp Request]
   RUNG wire#powerrail
      { S7_Templates := "SrcType := DInt" } EQ_Contact(in1 := "Unit1.Em4.ControlNodes".mainPnP.sequence.status.currentStep, in2 := #JOB_3_STEP_50)
      Contact( "Unit1.Em4.ControlNodes".mainPnP.sequence.status.seqActive )
      wire#w1
      Coil( "Unit1.Em4.ControlNodes".mainPnP."step".action1[350] )
   END_RUNG
   RUNG wire#w1
      Contact( "Unit1.Em4.ControlNodes".alignTable.jobInterface.loadJob2.loadingDone )
      Contact( "Unit1.EmNodes".emRelations.em06.sequence.Spare1.jobInterface[3].clampDone )
      Coil( "Unit1.Em4.ControlNodes".mainPnP."step".transition1[350] )
   END_RUNG
   RUNG wire#w1
      Contact( "Unit1.Em4.ControlNodes".mainPnP."step".transition1[350] )
      { S7_Templates := "time_type := Time" } #statTonTime[350].TON(pt := #delayTime, et =>)
      Move(in := #JOB_3_STEP_60, out1 => "Unit1.Em4.ControlNodes".mainPnP.sequence.status.nextStep)
   END_RUNG
   // the same network as SCL:
   "Unit1.Em4.ControlNodes".mainPnP."step".action1[350] := ("Unit1.Em4.ControlNodes".mainPnP.sequence.status.currentStep = #JOB_3_STEP_50) AND "Unit1.Em4.ControlNodes".mainPnP.sequence.status.seqActive;
   "Unit1.Em4.ControlNodes".mainPnP."step".transition1[350] := ("Unit1.Em4.ControlNodes".mainPnP.sequence.status.currentStep = #JOB_3_STEP_50) AND "Unit1.Em4.ControlNodes".mainPnP.sequence.status.seqActive AND "Unit1.Em4.ControlNodes".alignTable.jobInterface.loadJob2.loadingDone AND "Unit1.EmNodes".emRelations.em06.sequence.Spare1.jobInterface[3].clampDone;
   #statTonTime[350].TON(IN := ("Unit1.Em4.ControlNodes".mainPnP.sequence.status.currentStep = #JOB_3_STEP_50) AND "Unit1.Em4.ControlNodes".mainPnP.sequence.status.seqActive AND "Unit1.Em4.ControlNodes".mainPnP."step".transition1[350],
                         PT := #delayTime);
   IF #statTonTime[350].Q THEN
       "Unit1.Em4.ControlNodes".mainPnP.sequence.status.nextStep := #JOB_3_STEP_60;
   END_IF;
END_REGION

REGION Network 80: Step[360] : Main P&P 1.2 Vaccum Off
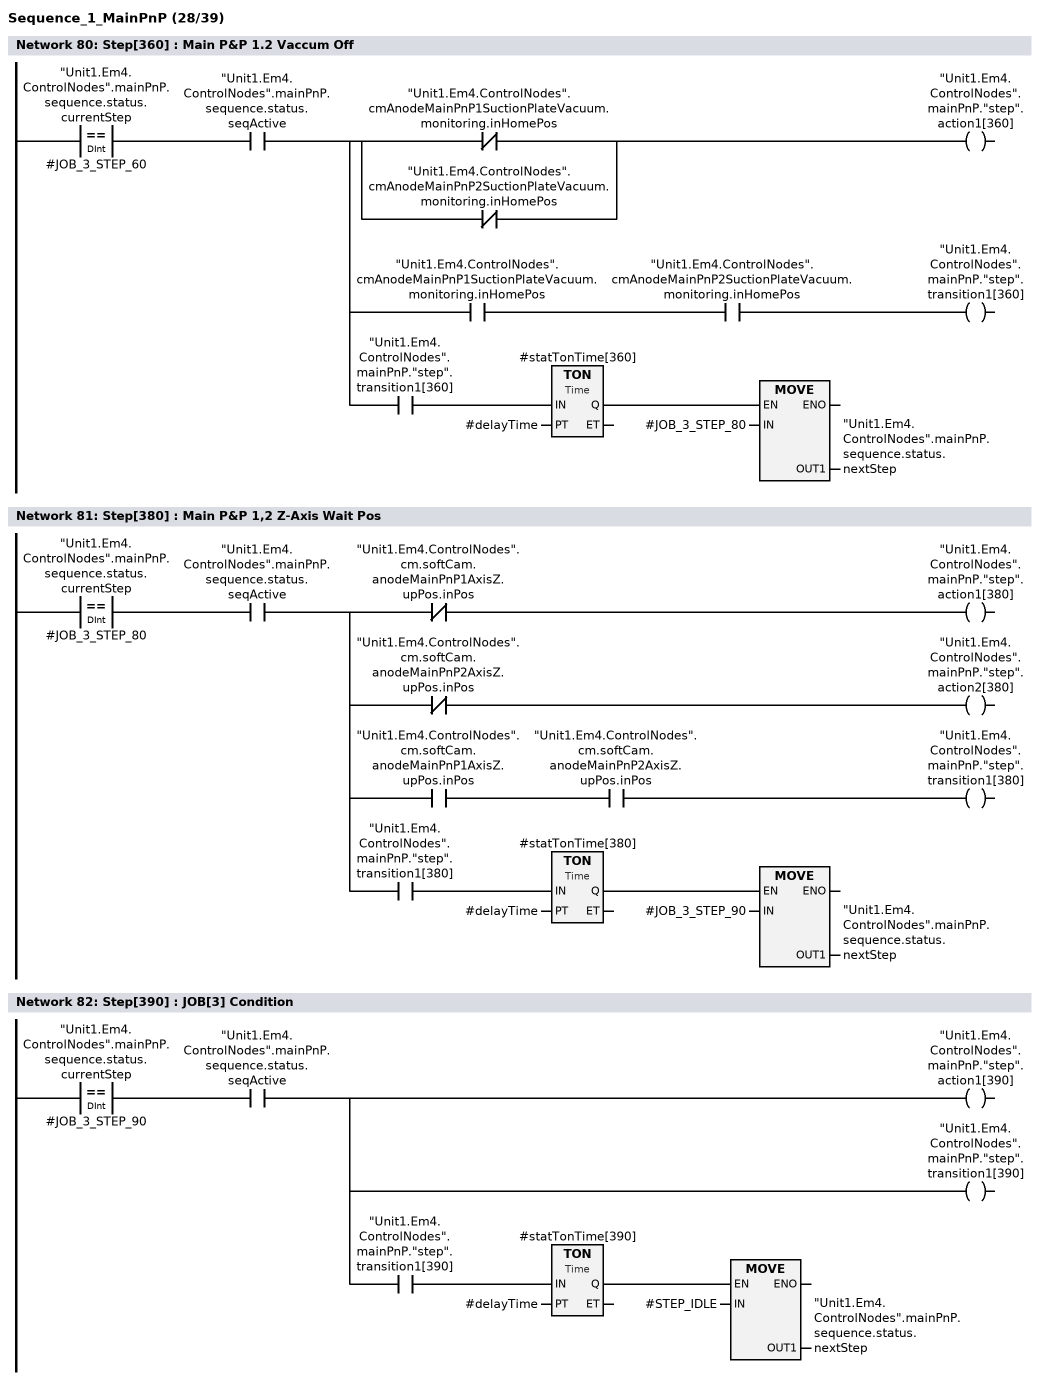
   RUNG wire#powerrail
      { S7_Templates := "SrcType := DInt" } EQ_Contact(in1 := "Unit1.Em4.ControlNodes".mainPnP.sequence.status.currentStep, in2 := #JOB_3_STEP_60)
      Contact( "Unit1.Em4.ControlNodes".mainPnP.sequence.status.seqActive )
      wire#w1
      I_Contact( "Unit1.Em4.ControlNodes".cmAnodeMainPnP1SuctionPlateVacuum.monitoring.inHomePos )
      wire#w2
      Coil( "Unit1.Em4.ControlNodes".mainPnP."step".action1[360] )
   END_RUNG
   RUNG wire#w1
      I_Contact( "Unit1.Em4.ControlNodes".cmAnodeMainPnP2SuctionPlateVacuum.monitoring.inHomePos )
   END_RUNG wire#w2
   RUNG wire#w1
      Contact( "Unit1.Em4.ControlNodes".cmAnodeMainPnP1SuctionPlateVacuum.monitoring.inHomePos )
      Contact( "Unit1.Em4.ControlNodes".cmAnodeMainPnP2SuctionPlateVacuum.monitoring.inHomePos )
      Coil( "Unit1.Em4.ControlNodes".mainPnP."step".transition1[360] )
   END_RUNG
   RUNG wire#w1
      Contact( "Unit1.Em4.ControlNodes".mainPnP."step".transition1[360] )
      { S7_Templates := "time_type := Time" } #statTonTime[360].TON(pt := #delayTime, et =>)
      Move(in := #JOB_3_STEP_80, out1 => "Unit1.Em4.ControlNodes".mainPnP.sequence.status.nextStep)
   END_RUNG
   // the same network as SCL:
   #_w1 := ("Unit1.Em4.ControlNodes".mainPnP.sequence.status.currentStep = #JOB_3_STEP_60) AND "Unit1.Em4.ControlNodes".mainPnP.sequence.status.seqActive;
   "Unit1.Em4.ControlNodes".mainPnP."step".action1[360] := #_w1 AND (NOT "Unit1.Em4.ControlNodes".cmAnodeMainPnP1SuctionPlateVacuum.monitoring.inHomePos OR NOT "Unit1.Em4.ControlNodes".cmAnodeMainPnP2SuctionPlateVacuum.monitoring.inHomePos);
   "Unit1.Em4.ControlNodes".mainPnP."step".transition1[360] := #_w1 AND "Unit1.Em4.ControlNodes".cmAnodeMainPnP1SuctionPlateVacuum.monitoring.inHomePos AND "Unit1.Em4.ControlNodes".cmAnodeMainPnP2SuctionPlateVacuum.monitoring.inHomePos;
   #statTonTime[360].TON(IN := #_w1 AND "Unit1.Em4.ControlNodes".mainPnP."step".transition1[360],
                         PT := #delayTime);
   IF #statTonTime[360].Q THEN
       "Unit1.Em4.ControlNodes".mainPnP.sequence.status.nextStep := #JOB_3_STEP_80;
   END_IF;
END_REGION

REGION Network 81: Step[380] : Main P&P 1,2 Z-Axis Wait Pos
   RUNG wire#powerrail
      { S7_Templates := "SrcType := DInt" } EQ_Contact(in1 := "Unit1.Em4.ControlNodes".mainPnP.sequence.status.currentStep, in2 := #JOB_3_STEP_80)
      Contact( "Unit1.Em4.ControlNodes".mainPnP.sequence.status.seqActive )
      wire#w1
      I_Contact( "Unit1.Em4.ControlNodes".cm.softCam.anodeMainPnP1AxisZ.upPos.inPos )
      Coil( "Unit1.Em4.ControlNodes".mainPnP."step".action1[380] )
   END_RUNG
   RUNG wire#w1
      I_Contact( "Unit1.Em4.ControlNodes".cm.softCam.anodeMainPnP2AxisZ.upPos.inPos )
      Coil( "Unit1.Em4.ControlNodes".mainPnP."step".action2[380] )
   END_RUNG
   RUNG wire#w1
      Contact( "Unit1.Em4.ControlNodes".cm.softCam.anodeMainPnP1AxisZ.upPos.inPos )
      Contact( "Unit1.Em4.ControlNodes".cm.softCam.anodeMainPnP2AxisZ.upPos.inPos )
      Coil( "Unit1.Em4.ControlNodes".mainPnP."step".transition1[380] )
   END_RUNG
   RUNG wire#w1
      Contact( "Unit1.Em4.ControlNodes".mainPnP."step".transition1[380] )
      { S7_Templates := "time_type := Time" } #statTonTime[380].TON(pt := #delayTime, et =>)
      Move(in := #JOB_3_STEP_90, out1 => "Unit1.Em4.ControlNodes".mainPnP.sequence.status.nextStep)
   END_RUNG
   // the same network as SCL:
   #_w1 := ("Unit1.Em4.ControlNodes".mainPnP.sequence.status.currentStep = #JOB_3_STEP_80) AND "Unit1.Em4.ControlNodes".mainPnP.sequence.status.seqActive;
   "Unit1.Em4.ControlNodes".mainPnP."step".action1[380] := #_w1 AND NOT "Unit1.Em4.ControlNodes".cm.softCam.anodeMainPnP1AxisZ.upPos.inPos;
   "Unit1.Em4.ControlNodes".mainPnP."step".action2[380] := #_w1 AND NOT "Unit1.Em4.ControlNodes".cm.softCam.anodeMainPnP2AxisZ.upPos.inPos;
   "Unit1.Em4.ControlNodes".mainPnP."step".transition1[380] := #_w1 AND "Unit1.Em4.ControlNodes".cm.softCam.anodeMainPnP1AxisZ.upPos.inPos AND "Unit1.Em4.ControlNodes".cm.softCam.anodeMainPnP2AxisZ.upPos.inPos;
   #statTonTime[380].TON(IN := #_w1 AND "Unit1.Em4.ControlNodes".mainPnP."step".transition1[380],
                         PT := #delayTime);
   IF #statTonTime[380].Q THEN
       "Unit1.Em4.ControlNodes".mainPnP.sequence.status.nextStep := #JOB_3_STEP_90;
   END_IF;
END_REGION

REGION Network 82: Step[390] : JOB[3] Condition
   RUNG wire#powerrail
      { S7_Templates := "SrcType := DInt" } EQ_Contact(in1 := "Unit1.Em4.ControlNodes".mainPnP.sequence.status.currentStep, in2 := #JOB_3_STEP_90)
      Contact( "Unit1.Em4.ControlNodes".mainPnP.sequence.status.seqActive )
      wire#w1
      Coil( "Unit1.Em4.ControlNodes".mainPnP."step".action1[390] )
   END_RUNG
   RUNG wire#w1
      Coil( "Unit1.Em4.ControlNodes".mainPnP."step".transition1[390] )
   END_RUNG
   RUNG wire#w1
      Contact( "Unit1.Em4.ControlNodes".mainPnP."step".transition1[390] )
      { S7_Templates := "time_type := Time" } #statTonTime[390].TON(pt := #delayTime, et =>)
      Move(in := #STEP_IDLE, out1 => "Unit1.Em4.ControlNodes".mainPnP.sequence.status.nextStep)
   END_RUNG
   // the same network as SCL:
   "Unit1.Em4.ControlNodes".mainPnP."step".action1[390] := ("Unit1.Em4.ControlNodes".mainPnP.sequence.status.currentStep = #JOB_3_STEP_90) AND "Unit1.Em4.ControlNodes".mainPnP.sequence.status.seqActive;
   "Unit1.Em4.ControlNodes".mainPnP."step".transition1[390] := ("Unit1.Em4.ControlNodes".mainPnP.sequence.status.currentStep = #JOB_3_STEP_90) AND "Unit1.Em4.ControlNodes".mainPnP.sequence.status.seqActive;
   #statTonTime[390].TON(IN := ("Unit1.Em4.ControlNodes".mainPnP.sequence.status.currentStep = #JOB_3_STEP_90) AND "Unit1.Em4.ControlNodes".mainPnP.sequence.status.seqActive AND "Unit1.Em4.ControlNodes".mainPnP."step".transition1[390],
                         PT := #delayTime);
   IF #statTonTime[390].Q THEN
       "Unit1.Em4.ControlNodes".mainPnP.sequence.status.nextStep := #STEP_IDLE;
   END_IF;
END_REGION

REGION Network 83: *************** JOB[4] Avoid ************************
END_REGION

REGION Network 84: Step[401] : JOB[4] Condition
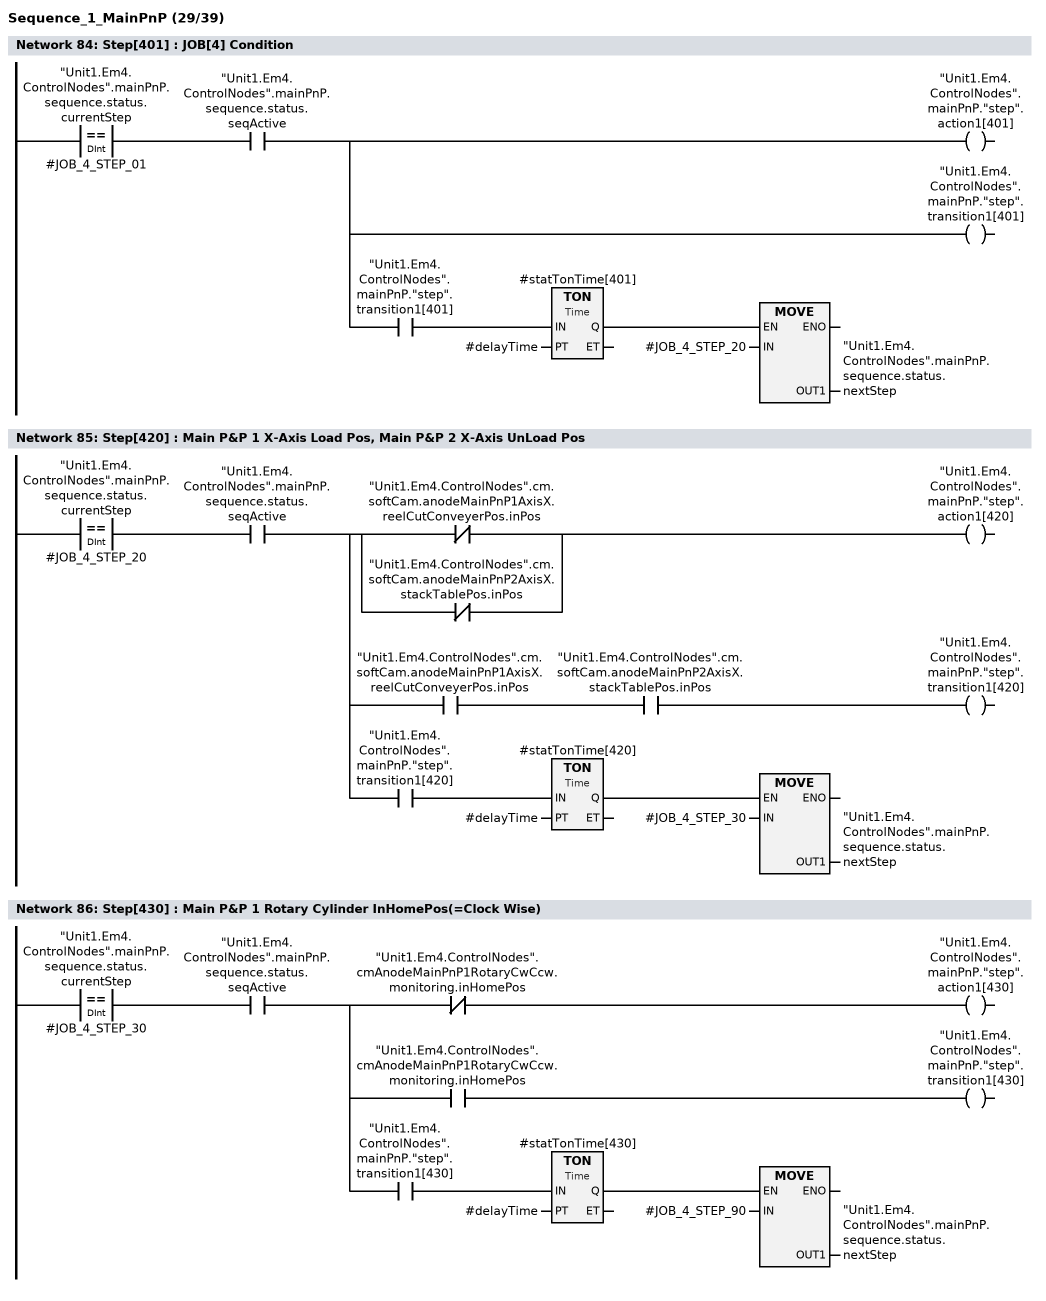
   RUNG wire#powerrail
      { S7_Templates := "SrcType := DInt" } EQ_Contact(in1 := "Unit1.Em4.ControlNodes".mainPnP.sequence.status.currentStep, in2 := #JOB_4_STEP_01)
      Contact( "Unit1.Em4.ControlNodes".mainPnP.sequence.status.seqActive )
      wire#w1
      Coil( "Unit1.Em4.ControlNodes".mainPnP."step".action1[401] )
   END_RUNG
   RUNG wire#w1
      Coil( "Unit1.Em4.ControlNodes".mainPnP."step".transition1[401] )
   END_RUNG
   RUNG wire#w1
      Contact( "Unit1.Em4.ControlNodes".mainPnP."step".transition1[401] )
      { S7_Templates := "time_type := Time" } #statTonTime[401].TON(pt := #delayTime, et =>)
      Move(in := #JOB_4_STEP_20, out1 => "Unit1.Em4.ControlNodes".mainPnP.sequence.status.nextStep)
   END_RUNG
   // the same network as SCL:
   "Unit1.Em4.ControlNodes".mainPnP."step".action1[401] := ("Unit1.Em4.ControlNodes".mainPnP.sequence.status.currentStep = #JOB_4_STEP_01) AND "Unit1.Em4.ControlNodes".mainPnP.sequence.status.seqActive;
   "Unit1.Em4.ControlNodes".mainPnP."step".transition1[401] := ("Unit1.Em4.ControlNodes".mainPnP.sequence.status.currentStep = #JOB_4_STEP_01) AND "Unit1.Em4.ControlNodes".mainPnP.sequence.status.seqActive;
   #statTonTime[401].TON(IN := ("Unit1.Em4.ControlNodes".mainPnP.sequence.status.currentStep = #JOB_4_STEP_01) AND "Unit1.Em4.ControlNodes".mainPnP.sequence.status.seqActive AND "Unit1.Em4.ControlNodes".mainPnP."step".transition1[401],
                         PT := #delayTime);
   IF #statTonTime[401].Q THEN
       "Unit1.Em4.ControlNodes".mainPnP.sequence.status.nextStep := #JOB_4_STEP_20;
   END_IF;
END_REGION

REGION Network 85: Step[420] : Main P&P 1 X-Axis Load Pos, Main P&P 2 X-Axis UnLoad Pos
   RUNG wire#powerrail
      { S7_Templates := "SrcType := DInt" } EQ_Contact(in1 := "Unit1.Em4.ControlNodes".mainPnP.sequence.status.currentStep, in2 := #JOB_4_STEP_20)
      Contact( "Unit1.Em4.ControlNodes".mainPnP.sequence.status.seqActive )
      wire#w1
      I_Contact( "Unit1.Em4.ControlNodes".cm.softCam.anodeMainPnP1AxisX.reelCutConveyerPos.inPos )
      wire#w2
      Coil( "Unit1.Em4.ControlNodes".mainPnP."step".action1[420] )
   END_RUNG
   RUNG wire#w1
      I_Contact( "Unit1.Em4.ControlNodes".cm.softCam.anodeMainPnP2AxisX.stackTablePos.inPos )
   END_RUNG wire#w2
   RUNG wire#w1
      Contact( "Unit1.Em4.ControlNodes".cm.softCam.anodeMainPnP1AxisX.reelCutConveyerPos.inPos )
      Contact( "Unit1.Em4.ControlNodes".cm.softCam.anodeMainPnP2AxisX.stackTablePos.inPos )
      Coil( "Unit1.Em4.ControlNodes".mainPnP."step".transition1[420] )
   END_RUNG
   RUNG wire#w1
      Contact( "Unit1.Em4.ControlNodes".mainPnP."step".transition1[420] )
      { S7_Templates := "time_type := Time" } #statTonTime[420].TON(pt := #delayTime, et =>)
      Move(in := #JOB_4_STEP_30, out1 => "Unit1.Em4.ControlNodes".mainPnP.sequence.status.nextStep)
   END_RUNG
   // the same network as SCL:
   #_w1 := ("Unit1.Em4.ControlNodes".mainPnP.sequence.status.currentStep = #JOB_4_STEP_20) AND "Unit1.Em4.ControlNodes".mainPnP.sequence.status.seqActive;
   "Unit1.Em4.ControlNodes".mainPnP."step".action1[420] := #_w1 AND (NOT "Unit1.Em4.ControlNodes".cm.softCam.anodeMainPnP1AxisX.reelCutConveyerPos.inPos OR NOT "Unit1.Em4.ControlNodes".cm.softCam.anodeMainPnP2AxisX.stackTablePos.inPos);
   "Unit1.Em4.ControlNodes".mainPnP."step".transition1[420] := #_w1 AND "Unit1.Em4.ControlNodes".cm.softCam.anodeMainPnP1AxisX.reelCutConveyerPos.inPos AND "Unit1.Em4.ControlNodes".cm.softCam.anodeMainPnP2AxisX.stackTablePos.inPos;
   #statTonTime[420].TON(IN := #_w1 AND "Unit1.Em4.ControlNodes".mainPnP."step".transition1[420],
                         PT := #delayTime);
   IF #statTonTime[420].Q THEN
       "Unit1.Em4.ControlNodes".mainPnP.sequence.status.nextStep := #JOB_4_STEP_30;
   END_IF;
END_REGION

REGION Network 86: Step[430] : Main P&P 1 Rotary Cylinder InHomePos(=Clock Wise)
   RUNG wire#powerrail
      { S7_Templates := "SrcType := DInt" } EQ_Contact(in1 := "Unit1.Em4.ControlNodes".mainPnP.sequence.status.currentStep, in2 := #JOB_4_STEP_30)
      Contact( "Unit1.Em4.ControlNodes".mainPnP.sequence.status.seqActive )
      wire#w1
      I_Contact( "Unit1.Em4.ControlNodes".cmAnodeMainPnP1RotaryCwCcw.monitoring.inHomePos )
      Coil( "Unit1.Em4.ControlNodes".mainPnP."step".action1[430] )
   END_RUNG
   RUNG wire#w1
      Contact( "Unit1.Em4.ControlNodes".cmAnodeMainPnP1RotaryCwCcw.monitoring.inHomePos )
      Coil( "Unit1.Em4.ControlNodes".mainPnP."step".transition1[430] )
   END_RUNG
   RUNG wire#w1
      Contact( "Unit1.Em4.ControlNodes".mainPnP."step".transition1[430] )
      { S7_Templates := "time_type := Time" } #statTonTime[430].TON(pt := #delayTime, et =>)
      Move(in := #JOB_4_STEP_90, out1 => "Unit1.Em4.ControlNodes".mainPnP.sequence.status.nextStep)
   END_RUNG
   // the same network as SCL:
   #_w1 := ("Unit1.Em4.ControlNodes".mainPnP.sequence.status.currentStep = #JOB_4_STEP_30) AND "Unit1.Em4.ControlNodes".mainPnP.sequence.status.seqActive;
   "Unit1.Em4.ControlNodes".mainPnP."step".action1[430] := #_w1 AND NOT "Unit1.Em4.ControlNodes".cmAnodeMainPnP1RotaryCwCcw.monitoring.inHomePos;
   "Unit1.Em4.ControlNodes".mainPnP."step".transition1[430] := #_w1 AND "Unit1.Em4.ControlNodes".cmAnodeMainPnP1RotaryCwCcw.monitoring.inHomePos;
   #statTonTime[430].TON(IN := #_w1 AND "Unit1.Em4.ControlNodes".mainPnP."step".transition1[430],
                         PT := #delayTime);
   IF #statTonTime[430].Q THEN
       "Unit1.Em4.ControlNodes".mainPnP.sequence.status.nextStep := #JOB_4_STEP_90;
   END_IF;
END_REGION

REGION Network 87: Step[490] : JOB[4] Condition
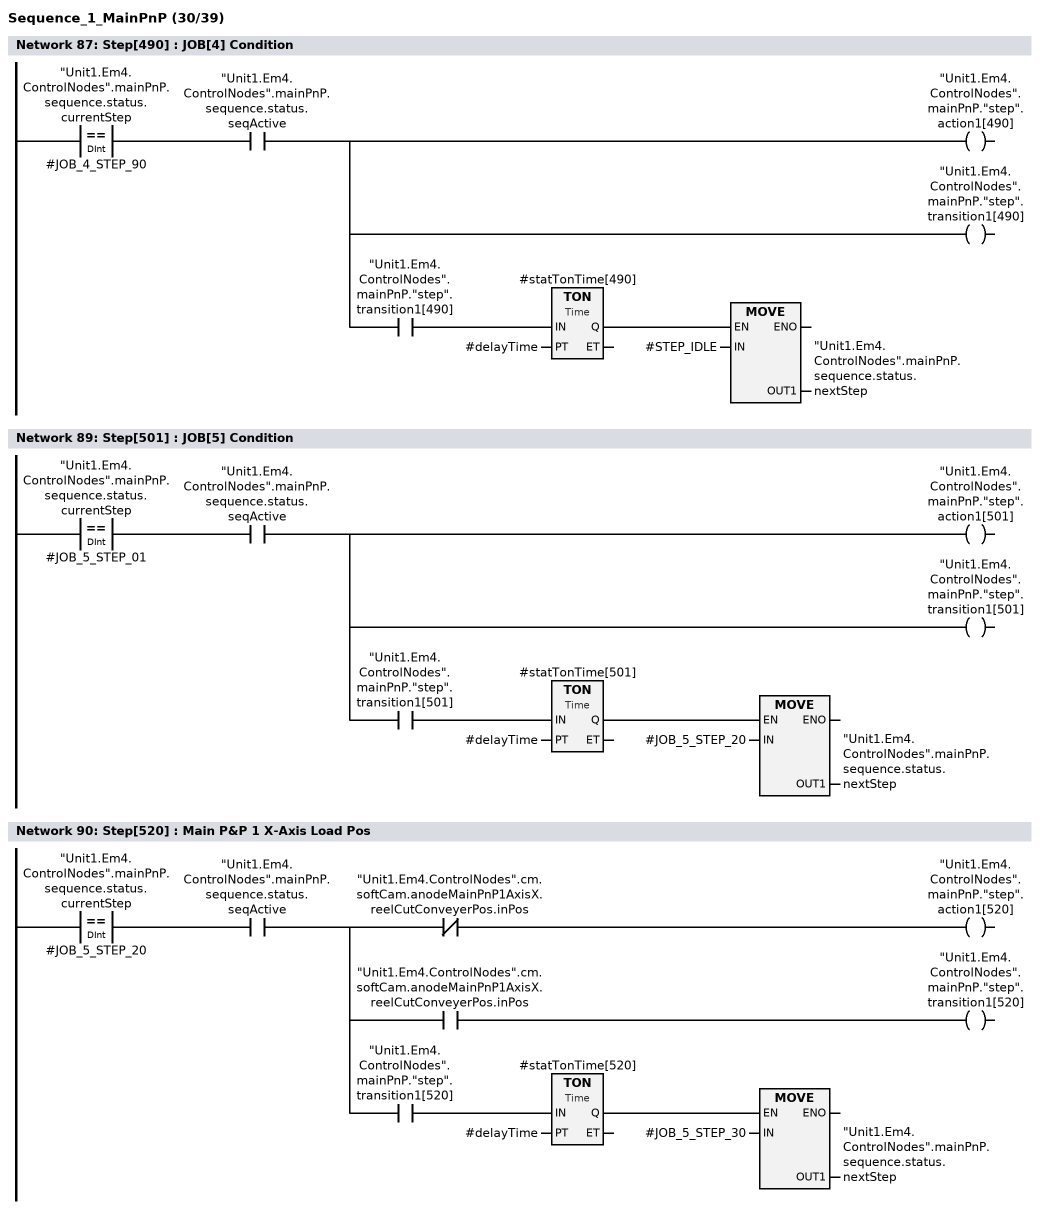
   RUNG wire#powerrail
      { S7_Templates := "SrcType := DInt" } EQ_Contact(in1 := "Unit1.Em4.ControlNodes".mainPnP.sequence.status.currentStep, in2 := #JOB_4_STEP_90)
      Contact( "Unit1.Em4.ControlNodes".mainPnP.sequence.status.seqActive )
      wire#w1
      Coil( "Unit1.Em4.ControlNodes".mainPnP."step".action1[490] )
   END_RUNG
   RUNG wire#w1
      Coil( "Unit1.Em4.ControlNodes".mainPnP."step".transition1[490] )
   END_RUNG
   RUNG wire#w1
      Contact( "Unit1.Em4.ControlNodes".mainPnP."step".transition1[490] )
      { S7_Templates := "time_type := Time" } #statTonTime[490].TON(pt := #delayTime, et =>)
      Move(in := #STEP_IDLE, out1 => "Unit1.Em4.ControlNodes".mainPnP.sequence.status.nextStep)
   END_RUNG
   // the same network as SCL:
   "Unit1.Em4.ControlNodes".mainPnP."step".action1[490] := ("Unit1.Em4.ControlNodes".mainPnP.sequence.status.currentStep = #JOB_4_STEP_90) AND "Unit1.Em4.ControlNodes".mainPnP.sequence.status.seqActive;
   "Unit1.Em4.ControlNodes".mainPnP."step".transition1[490] := ("Unit1.Em4.ControlNodes".mainPnP.sequence.status.currentStep = #JOB_4_STEP_90) AND "Unit1.Em4.ControlNodes".mainPnP.sequence.status.seqActive;
   #statTonTime[490].TON(IN := ("Unit1.Em4.ControlNodes".mainPnP.sequence.status.currentStep = #JOB_4_STEP_90) AND "Unit1.Em4.ControlNodes".mainPnP.sequence.status.seqActive AND "Unit1.Em4.ControlNodes".mainPnP."step".transition1[490],
                         PT := #delayTime);
   IF #statTonTime[490].Q THEN
       "Unit1.Em4.ControlNodes".mainPnP.sequence.status.nextStep := #STEP_IDLE;
   END_IF;
END_REGION

REGION Network 88: *************** JOB[5] One Loading ************************
END_REGION

REGION Network 89: Step[501] : JOB[5] Condition
   RUNG wire#powerrail
      { S7_Templates := "SrcType := DInt" } EQ_Contact(in1 := "Unit1.Em4.ControlNodes".mainPnP.sequence.status.currentStep, in2 := #JOB_5_STEP_01)
      Contact( "Unit1.Em4.ControlNodes".mainPnP.sequence.status.seqActive )
      wire#w1
      Coil( "Unit1.Em4.ControlNodes".mainPnP."step".action1[501] )
   END_RUNG
   RUNG wire#w1
      Coil( "Unit1.Em4.ControlNodes".mainPnP."step".transition1[501] )
   END_RUNG
   RUNG wire#w1
      Contact( "Unit1.Em4.ControlNodes".mainPnP."step".transition1[501] )
      { S7_Templates := "time_type := Time" } #statTonTime[501].TON(pt := #delayTime, et =>)
      Move(in := #JOB_5_STEP_20, out1 => "Unit1.Em4.ControlNodes".mainPnP.sequence.status.nextStep)
   END_RUNG
   // the same network as SCL:
   "Unit1.Em4.ControlNodes".mainPnP."step".action1[501] := ("Unit1.Em4.ControlNodes".mainPnP.sequence.status.currentStep = #JOB_5_STEP_01) AND "Unit1.Em4.ControlNodes".mainPnP.sequence.status.seqActive;
   "Unit1.Em4.ControlNodes".mainPnP."step".transition1[501] := ("Unit1.Em4.ControlNodes".mainPnP.sequence.status.currentStep = #JOB_5_STEP_01) AND "Unit1.Em4.ControlNodes".mainPnP.sequence.status.seqActive;
   #statTonTime[501].TON(IN := ("Unit1.Em4.ControlNodes".mainPnP.sequence.status.currentStep = #JOB_5_STEP_01) AND "Unit1.Em4.ControlNodes".mainPnP.sequence.status.seqActive AND "Unit1.Em4.ControlNodes".mainPnP."step".transition1[501],
                         PT := #delayTime);
   IF #statTonTime[501].Q THEN
       "Unit1.Em4.ControlNodes".mainPnP.sequence.status.nextStep := #JOB_5_STEP_20;
   END_IF;
END_REGION

REGION Network 90: Step[520] : Main P&P 1 X-Axis Load Pos
   RUNG wire#powerrail
      { S7_Templates := "SrcType := DInt" } EQ_Contact(in1 := "Unit1.Em4.ControlNodes".mainPnP.sequence.status.currentStep, in2 := #JOB_5_STEP_20)
      Contact( "Unit1.Em4.ControlNodes".mainPnP.sequence.status.seqActive )
      wire#w1
      I_Contact( "Unit1.Em4.ControlNodes".cm.softCam.anodeMainPnP1AxisX.reelCutConveyerPos.inPos )
      Coil( "Unit1.Em4.ControlNodes".mainPnP."step".action1[520] )
   END_RUNG
   RUNG wire#w1
      Contact( "Unit1.Em4.ControlNodes".cm.softCam.anodeMainPnP1AxisX.reelCutConveyerPos.inPos )
      Coil( "Unit1.Em4.ControlNodes".mainPnP."step".transition1[520] )
   END_RUNG
   RUNG wire#w1
      Contact( "Unit1.Em4.ControlNodes".mainPnP."step".transition1[520] )
      { S7_Templates := "time_type := Time" } #statTonTime[520].TON(pt := #delayTime, et =>)
      Move(in := #JOB_5_STEP_30, out1 => "Unit1.Em4.ControlNodes".mainPnP.sequence.status.nextStep)
   END_RUNG
   // the same network as SCL:
   #_w1 := ("Unit1.Em4.ControlNodes".mainPnP.sequence.status.currentStep = #JOB_5_STEP_20) AND "Unit1.Em4.ControlNodes".mainPnP.sequence.status.seqActive;
   "Unit1.Em4.ControlNodes".mainPnP."step".action1[520] := #_w1 AND NOT "Unit1.Em4.ControlNodes".cm.softCam.anodeMainPnP1AxisX.reelCutConveyerPos.inPos;
   "Unit1.Em4.ControlNodes".mainPnP."step".transition1[520] := #_w1 AND "Unit1.Em4.ControlNodes".cm.softCam.anodeMainPnP1AxisX.reelCutConveyerPos.inPos;
   #statTonTime[520].TON(IN := #_w1 AND "Unit1.Em4.ControlNodes".mainPnP."step".transition1[520],
                         PT := #delayTime);
   IF #statTonTime[520].Q THEN
       "Unit1.Em4.ControlNodes".mainPnP.sequence.status.nextStep := #JOB_5_STEP_30;
   END_IF;
END_REGION

REGION Network 91: Step[530] : Main P&P 1 Rotary Cylinder InHomePos
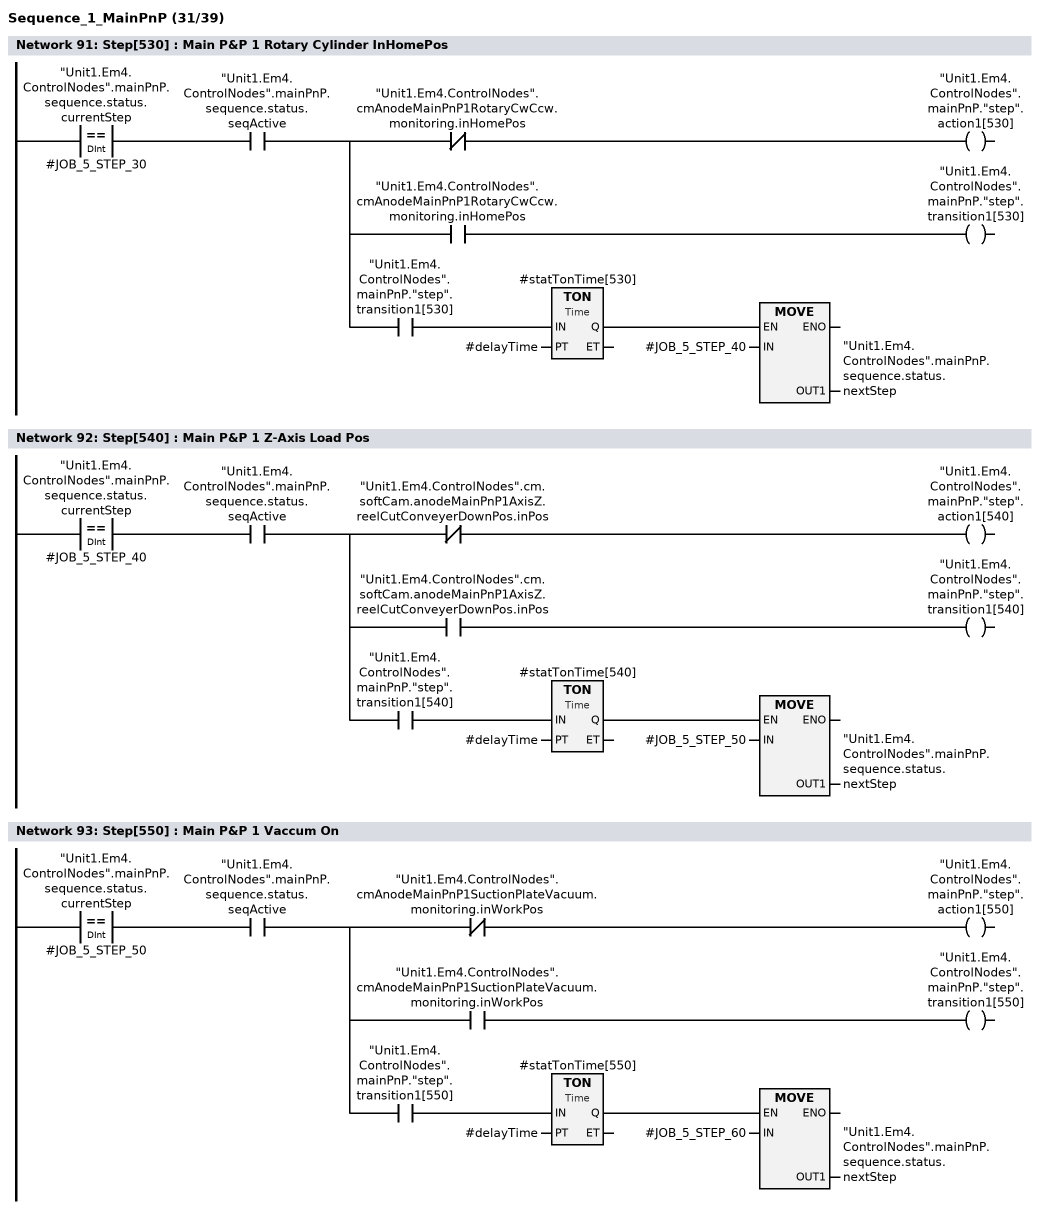
   RUNG wire#powerrail
      { S7_Templates := "SrcType := DInt" } EQ_Contact(in1 := "Unit1.Em4.ControlNodes".mainPnP.sequence.status.currentStep, in2 := #JOB_5_STEP_30)
      Contact( "Unit1.Em4.ControlNodes".mainPnP.sequence.status.seqActive )
      wire#w1
      I_Contact( "Unit1.Em4.ControlNodes".cmAnodeMainPnP1RotaryCwCcw.monitoring.inHomePos )
      Coil( "Unit1.Em4.ControlNodes".mainPnP."step".action1[530] )
   END_RUNG
   RUNG wire#w1
      Contact( "Unit1.Em4.ControlNodes".cmAnodeMainPnP1RotaryCwCcw.monitoring.inHomePos )
      Coil( "Unit1.Em4.ControlNodes".mainPnP."step".transition1[530] )
   END_RUNG
   RUNG wire#w1
      Contact( "Unit1.Em4.ControlNodes".mainPnP."step".transition1[530] )
      { S7_Templates := "time_type := Time" } #statTonTime[530].TON(pt := #delayTime, et =>)
      Move(in := #JOB_5_STEP_40, out1 => "Unit1.Em4.ControlNodes".mainPnP.sequence.status.nextStep)
   END_RUNG
   // the same network as SCL:
   #_w1 := ("Unit1.Em4.ControlNodes".mainPnP.sequence.status.currentStep = #JOB_5_STEP_30) AND "Unit1.Em4.ControlNodes".mainPnP.sequence.status.seqActive;
   "Unit1.Em4.ControlNodes".mainPnP."step".action1[530] := #_w1 AND NOT "Unit1.Em4.ControlNodes".cmAnodeMainPnP1RotaryCwCcw.monitoring.inHomePos;
   "Unit1.Em4.ControlNodes".mainPnP."step".transition1[530] := #_w1 AND "Unit1.Em4.ControlNodes".cmAnodeMainPnP1RotaryCwCcw.monitoring.inHomePos;
   #statTonTime[530].TON(IN := #_w1 AND "Unit1.Em4.ControlNodes".mainPnP."step".transition1[530],
                         PT := #delayTime);
   IF #statTonTime[530].Q THEN
       "Unit1.Em4.ControlNodes".mainPnP.sequence.status.nextStep := #JOB_5_STEP_40;
   END_IF;
END_REGION

REGION Network 92: Step[540] : Main P&P 1 Z-Axis Load Pos
   RUNG wire#powerrail
      { S7_Templates := "SrcType := DInt" } EQ_Contact(in1 := "Unit1.Em4.ControlNodes".mainPnP.sequence.status.currentStep, in2 := #JOB_5_STEP_40)
      Contact( "Unit1.Em4.ControlNodes".mainPnP.sequence.status.seqActive )
      wire#w1
      I_Contact( "Unit1.Em4.ControlNodes".cm.softCam.anodeMainPnP1AxisZ.reelCutConveyerDownPos.inPos )
      Coil( "Unit1.Em4.ControlNodes".mainPnP."step".action1[540] )
   END_RUNG
   RUNG wire#w1
      Contact( "Unit1.Em4.ControlNodes".cm.softCam.anodeMainPnP1AxisZ.reelCutConveyerDownPos.inPos )
      Coil( "Unit1.Em4.ControlNodes".mainPnP."step".transition1[540] )
   END_RUNG
   RUNG wire#w1
      Contact( "Unit1.Em4.ControlNodes".mainPnP."step".transition1[540] )
      { S7_Templates := "time_type := Time" } #statTonTime[540].TON(pt := #delayTime, et =>)
      Move(in := #JOB_5_STEP_50, out1 => "Unit1.Em4.ControlNodes".mainPnP.sequence.status.nextStep)
   END_RUNG
   // the same network as SCL:
   #_w1 := ("Unit1.Em4.ControlNodes".mainPnP.sequence.status.currentStep = #JOB_5_STEP_40) AND "Unit1.Em4.ControlNodes".mainPnP.sequence.status.seqActive;
   "Unit1.Em4.ControlNodes".mainPnP."step".action1[540] := #_w1 AND NOT "Unit1.Em4.ControlNodes".cm.softCam.anodeMainPnP1AxisZ.reelCutConveyerDownPos.inPos;
   "Unit1.Em4.ControlNodes".mainPnP."step".transition1[540] := #_w1 AND "Unit1.Em4.ControlNodes".cm.softCam.anodeMainPnP1AxisZ.reelCutConveyerDownPos.inPos;
   #statTonTime[540].TON(IN := #_w1 AND "Unit1.Em4.ControlNodes".mainPnP."step".transition1[540],
                         PT := #delayTime);
   IF #statTonTime[540].Q THEN
       "Unit1.Em4.ControlNodes".mainPnP.sequence.status.nextStep := #JOB_5_STEP_50;
   END_IF;
END_REGION

REGION Network 93: Step[550] : Main P&P 1 Vaccum On
   RUNG wire#powerrail
      { S7_Templates := "SrcType := DInt" } EQ_Contact(in1 := "Unit1.Em4.ControlNodes".mainPnP.sequence.status.currentStep, in2 := #JOB_5_STEP_50)
      Contact( "Unit1.Em4.ControlNodes".mainPnP.sequence.status.seqActive )
      wire#w1
      I_Contact( "Unit1.Em4.ControlNodes".cmAnodeMainPnP1SuctionPlateVacuum.monitoring.inWorkPos )
      Coil( "Unit1.Em4.ControlNodes".mainPnP."step".action1[550] )
   END_RUNG
   RUNG wire#w1
      Contact( "Unit1.Em4.ControlNodes".cmAnodeMainPnP1SuctionPlateVacuum.monitoring.inWorkPos )
      Coil( "Unit1.Em4.ControlNodes".mainPnP."step".transition1[550] )
   END_RUNG
   RUNG wire#w1
      Contact( "Unit1.Em4.ControlNodes".mainPnP."step".transition1[550] )
      { S7_Templates := "time_type := Time" } #statTonTime[550].TON(pt := #delayTime, et =>)
      Move(in := #JOB_5_STEP_60, out1 => "Unit1.Em4.ControlNodes".mainPnP.sequence.status.nextStep)
   END_RUNG
   // the same network as SCL:
   #_w1 := ("Unit1.Em4.ControlNodes".mainPnP.sequence.status.currentStep = #JOB_5_STEP_50) AND "Unit1.Em4.ControlNodes".mainPnP.sequence.status.seqActive;
   "Unit1.Em4.ControlNodes".mainPnP."step".action1[550] := #_w1 AND NOT "Unit1.Em4.ControlNodes".cmAnodeMainPnP1SuctionPlateVacuum.monitoring.inWorkPos;
   "Unit1.Em4.ControlNodes".mainPnP."step".transition1[550] := #_w1 AND "Unit1.Em4.ControlNodes".cmAnodeMainPnP1SuctionPlateVacuum.monitoring.inWorkPos;
   #statTonTime[550].TON(IN := #_w1 AND "Unit1.Em4.ControlNodes".mainPnP."step".transition1[550],
                         PT := #delayTime);
   IF #statTonTime[550].Q THEN
       "Unit1.Em4.ControlNodes".mainPnP.sequence.status.nextStep := #JOB_5_STEP_60;
   END_IF;
END_REGION

REGION Network 94: Step[560] : Main P&P 1 Pick Up Blow On
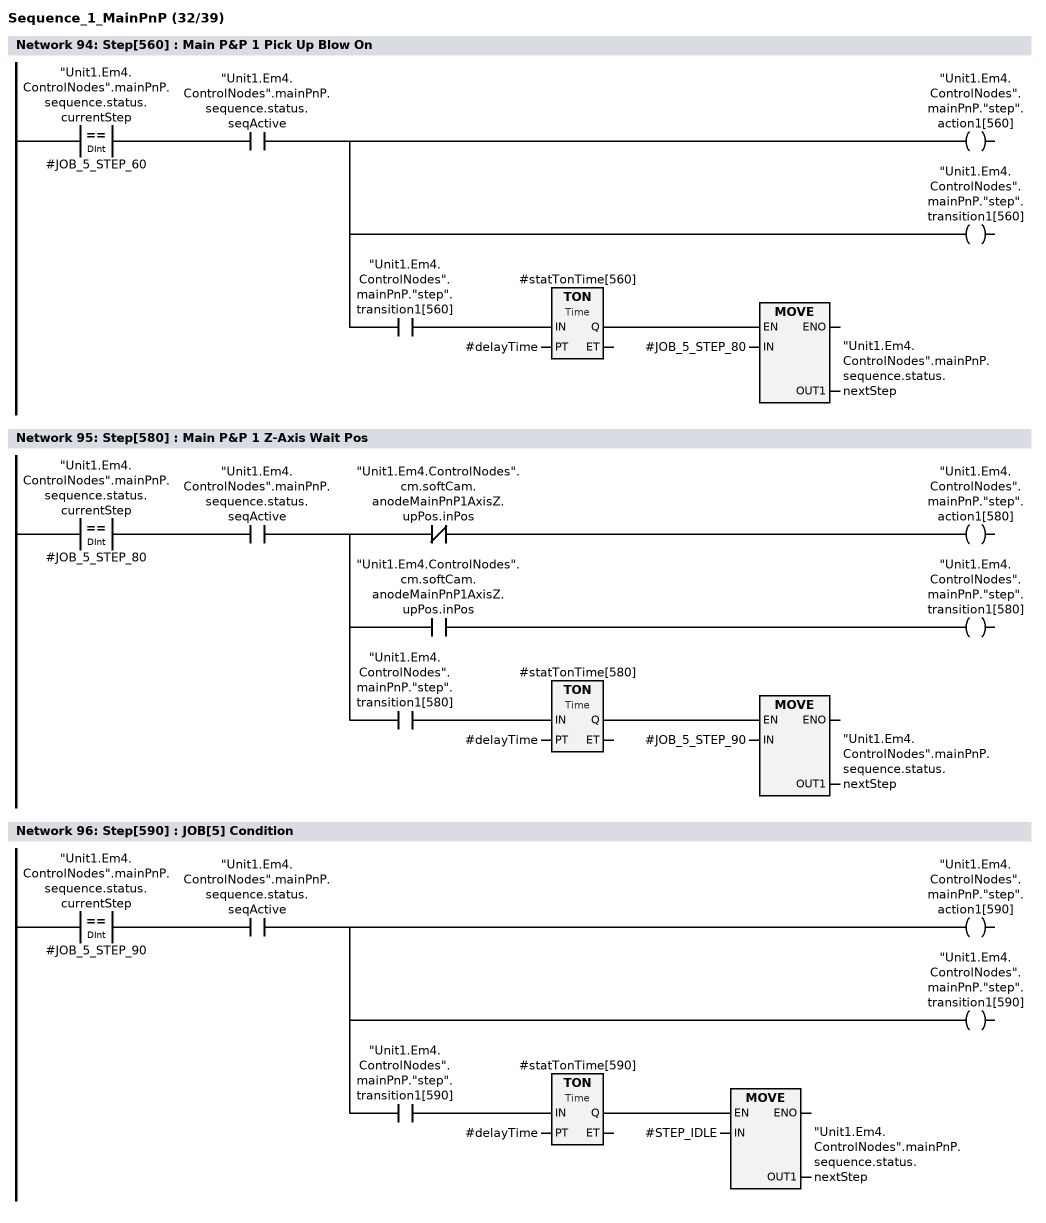
   RUNG wire#powerrail
      { S7_Templates := "SrcType := DInt" } EQ_Contact(in1 := "Unit1.Em4.ControlNodes".mainPnP.sequence.status.currentStep, in2 := #JOB_5_STEP_60)
      Contact( "Unit1.Em4.ControlNodes".mainPnP.sequence.status.seqActive )
      wire#w1
      Coil( "Unit1.Em4.ControlNodes".mainPnP."step".action1[560] )
   END_RUNG
   RUNG wire#w1
      Coil( "Unit1.Em4.ControlNodes".mainPnP."step".transition1[560] )
   END_RUNG
   RUNG wire#w1
      Contact( "Unit1.Em4.ControlNodes".mainPnP."step".transition1[560] )
      { S7_Templates := "time_type := Time" } #statTonTime[560].TON(pt := #delayTime, et =>)
      Move(in := #JOB_5_STEP_80, out1 => "Unit1.Em4.ControlNodes".mainPnP.sequence.status.nextStep)
   END_RUNG
   // the same network as SCL:
   "Unit1.Em4.ControlNodes".mainPnP."step".action1[560] := ("Unit1.Em4.ControlNodes".mainPnP.sequence.status.currentStep = #JOB_5_STEP_60) AND "Unit1.Em4.ControlNodes".mainPnP.sequence.status.seqActive;
   "Unit1.Em4.ControlNodes".mainPnP."step".transition1[560] := ("Unit1.Em4.ControlNodes".mainPnP.sequence.status.currentStep = #JOB_5_STEP_60) AND "Unit1.Em4.ControlNodes".mainPnP.sequence.status.seqActive;
   #statTonTime[560].TON(IN := ("Unit1.Em4.ControlNodes".mainPnP.sequence.status.currentStep = #JOB_5_STEP_60) AND "Unit1.Em4.ControlNodes".mainPnP.sequence.status.seqActive AND "Unit1.Em4.ControlNodes".mainPnP."step".transition1[560],
                         PT := #delayTime);
   IF #statTonTime[560].Q THEN
       "Unit1.Em4.ControlNodes".mainPnP.sequence.status.nextStep := #JOB_5_STEP_80;
   END_IF;
END_REGION

REGION Network 95: Step[580] : Main P&P 1 Z-Axis Wait Pos
   RUNG wire#powerrail
      { S7_Templates := "SrcType := DInt" } EQ_Contact(in1 := "Unit1.Em4.ControlNodes".mainPnP.sequence.status.currentStep, in2 := #JOB_5_STEP_80)
      Contact( "Unit1.Em4.ControlNodes".mainPnP.sequence.status.seqActive )
      wire#w1
      I_Contact( "Unit1.Em4.ControlNodes".cm.softCam.anodeMainPnP1AxisZ.upPos.inPos )
      Coil( "Unit1.Em4.ControlNodes".mainPnP."step".action1[580] )
   END_RUNG
   RUNG wire#w1
      Contact( "Unit1.Em4.ControlNodes".cm.softCam.anodeMainPnP1AxisZ.upPos.inPos )
      Coil( "Unit1.Em4.ControlNodes".mainPnP."step".transition1[580] )
   END_RUNG
   RUNG wire#w1
      Contact( "Unit1.Em4.ControlNodes".mainPnP."step".transition1[580] )
      { S7_Templates := "time_type := Time" } #statTonTime[580].TON(pt := #delayTime, et =>)
      Move(in := #JOB_5_STEP_90, out1 => "Unit1.Em4.ControlNodes".mainPnP.sequence.status.nextStep)
   END_RUNG
   // the same network as SCL:
   #_w1 := ("Unit1.Em4.ControlNodes".mainPnP.sequence.status.currentStep = #JOB_5_STEP_80) AND "Unit1.Em4.ControlNodes".mainPnP.sequence.status.seqActive;
   "Unit1.Em4.ControlNodes".mainPnP."step".action1[580] := #_w1 AND NOT "Unit1.Em4.ControlNodes".cm.softCam.anodeMainPnP1AxisZ.upPos.inPos;
   "Unit1.Em4.ControlNodes".mainPnP."step".transition1[580] := #_w1 AND "Unit1.Em4.ControlNodes".cm.softCam.anodeMainPnP1AxisZ.upPos.inPos;
   #statTonTime[580].TON(IN := #_w1 AND "Unit1.Em4.ControlNodes".mainPnP."step".transition1[580],
                         PT := #delayTime);
   IF #statTonTime[580].Q THEN
       "Unit1.Em4.ControlNodes".mainPnP.sequence.status.nextStep := #JOB_5_STEP_90;
   END_IF;
END_REGION

REGION Network 96: Step[590] : JOB[5] Condition
   RUNG wire#powerrail
      { S7_Templates := "SrcType := DInt" } EQ_Contact(in1 := "Unit1.Em4.ControlNodes".mainPnP.sequence.status.currentStep, in2 := #JOB_5_STEP_90)
      Contact( "Unit1.Em4.ControlNodes".mainPnP.sequence.status.seqActive )
      wire#w1
      Coil( "Unit1.Em4.ControlNodes".mainPnP."step".action1[590] )
   END_RUNG
   RUNG wire#w1
      Coil( "Unit1.Em4.ControlNodes".mainPnP."step".transition1[590] )
   END_RUNG
   RUNG wire#w1
      Contact( "Unit1.Em4.ControlNodes".mainPnP."step".transition1[590] )
      { S7_Templates := "time_type := Time" } #statTonTime[590].TON(pt := #delayTime, et =>)
      Move(in := #STEP_IDLE, out1 => "Unit1.Em4.ControlNodes".mainPnP.sequence.status.nextStep)
   END_RUNG
   // the same network as SCL:
   "Unit1.Em4.ControlNodes".mainPnP."step".action1[590] := ("Unit1.Em4.ControlNodes".mainPnP.sequence.status.currentStep = #JOB_5_STEP_90) AND "Unit1.Em4.ControlNodes".mainPnP.sequence.status.seqActive;
   "Unit1.Em4.ControlNodes".mainPnP."step".transition1[590] := ("Unit1.Em4.ControlNodes".mainPnP.sequence.status.currentStep = #JOB_5_STEP_90) AND "Unit1.Em4.ControlNodes".mainPnP.sequence.status.seqActive;
   #statTonTime[590].TON(IN := ("Unit1.Em4.ControlNodes".mainPnP.sequence.status.currentStep = #JOB_5_STEP_90) AND "Unit1.Em4.ControlNodes".mainPnP.sequence.status.seqActive AND "Unit1.Em4.ControlNodes".mainPnP."step".transition1[590],
                         PT := #delayTime);
   IF #statTonTime[590].Q THEN
       "Unit1.Em4.ControlNodes".mainPnP.sequence.status.nextStep := #STEP_IDLE;
   END_IF;
END_REGION

REGION Network 97: *************** JOB[6] One UnLoading ************************
END_REGION

REGION Network 98: Step[601] : JOB[6] Condition
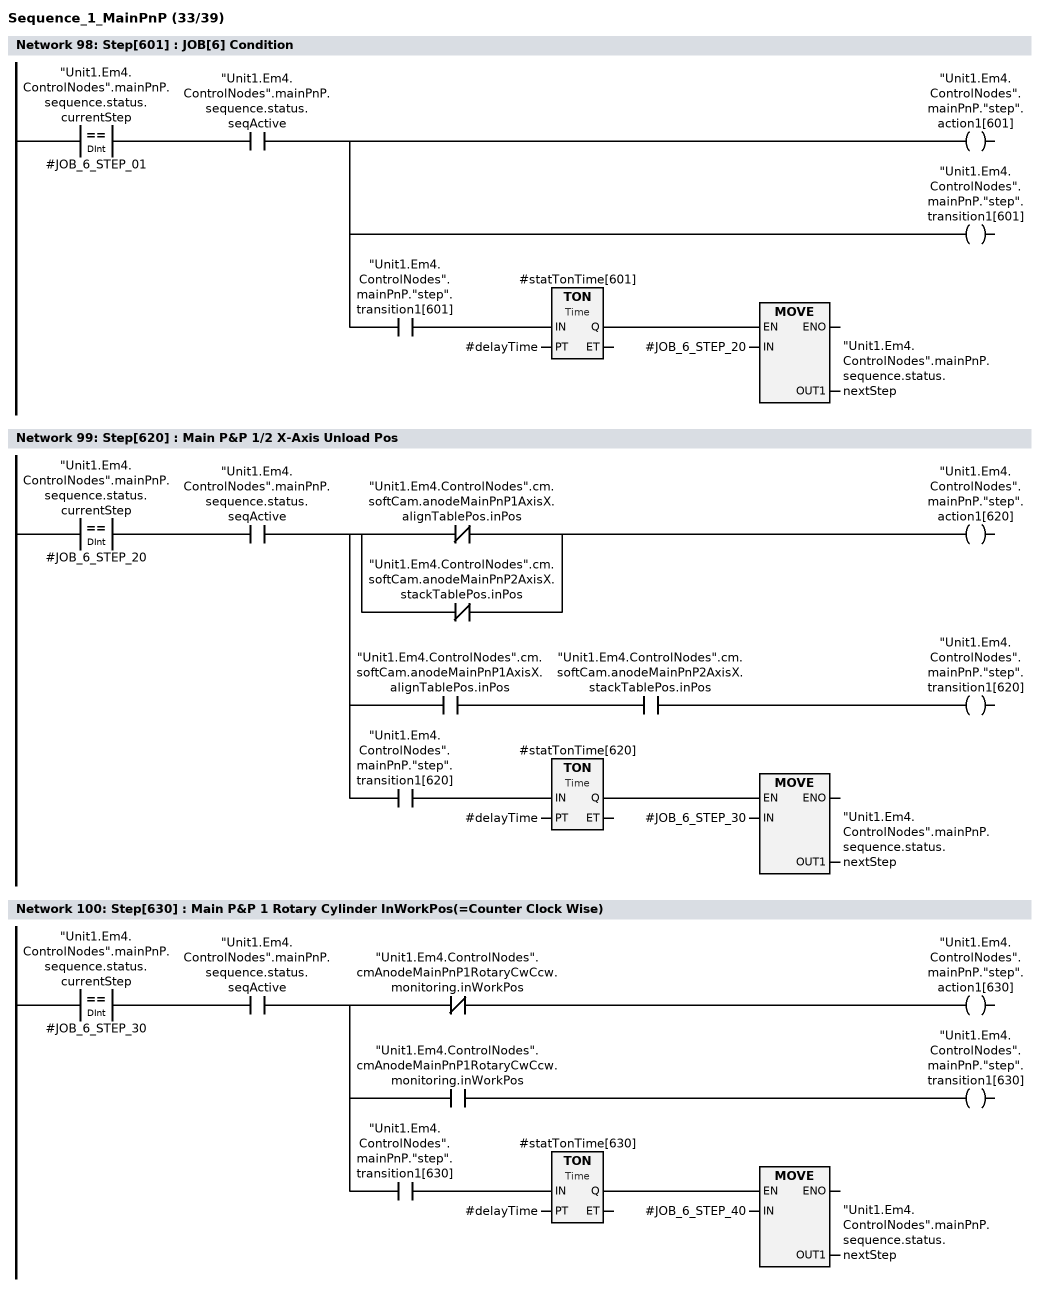
   RUNG wire#powerrail
      { S7_Templates := "SrcType := DInt" } EQ_Contact(in1 := "Unit1.Em4.ControlNodes".mainPnP.sequence.status.currentStep, in2 := #JOB_6_STEP_01)
      Contact( "Unit1.Em4.ControlNodes".mainPnP.sequence.status.seqActive )
      wire#w1
      Coil( "Unit1.Em4.ControlNodes".mainPnP."step".action1[601] )
   END_RUNG
   RUNG wire#w1
      Coil( "Unit1.Em4.ControlNodes".mainPnP."step".transition1[601] )
   END_RUNG
   RUNG wire#w1
      Contact( "Unit1.Em4.ControlNodes".mainPnP."step".transition1[601] )
      { S7_Templates := "time_type := Time" } #statTonTime[601].TON(pt := #delayTime, et =>)
      Move(in := #JOB_6_STEP_20, out1 => "Unit1.Em4.ControlNodes".mainPnP.sequence.status.nextStep)
   END_RUNG
   // the same network as SCL:
   "Unit1.Em4.ControlNodes".mainPnP."step".action1[601] := ("Unit1.Em4.ControlNodes".mainPnP.sequence.status.currentStep = #JOB_6_STEP_01) AND "Unit1.Em4.ControlNodes".mainPnP.sequence.status.seqActive;
   "Unit1.Em4.ControlNodes".mainPnP."step".transition1[601] := ("Unit1.Em4.ControlNodes".mainPnP.sequence.status.currentStep = #JOB_6_STEP_01) AND "Unit1.Em4.ControlNodes".mainPnP.sequence.status.seqActive;
   #statTonTime[601].TON(IN := ("Unit1.Em4.ControlNodes".mainPnP.sequence.status.currentStep = #JOB_6_STEP_01) AND "Unit1.Em4.ControlNodes".mainPnP.sequence.status.seqActive AND "Unit1.Em4.ControlNodes".mainPnP."step".transition1[601],
                         PT := #delayTime);
   IF #statTonTime[601].Q THEN
       "Unit1.Em4.ControlNodes".mainPnP.sequence.status.nextStep := #JOB_6_STEP_20;
   END_IF;
END_REGION

REGION Network 99: Step[620] : Main P&P 1/2 X-Axis Unload Pos
   RUNG wire#powerrail
      { S7_Templates := "SrcType := DInt" } EQ_Contact(in1 := "Unit1.Em4.ControlNodes".mainPnP.sequence.status.currentStep, in2 := #JOB_6_STEP_20)
      Contact( "Unit1.Em4.ControlNodes".mainPnP.sequence.status.seqActive )
      wire#w1
      I_Contact( "Unit1.Em4.ControlNodes".cm.softCam.anodeMainPnP1AxisX.alignTablePos.inPos )
      wire#w2
      Coil( "Unit1.Em4.ControlNodes".mainPnP."step".action1[620] )
   END_RUNG
   RUNG wire#w1
      I_Contact( "Unit1.Em4.ControlNodes".cm.softCam.anodeMainPnP2AxisX.stackTablePos.inPos )
   END_RUNG wire#w2
   RUNG wire#w1
      Contact( "Unit1.Em4.ControlNodes".cm.softCam.anodeMainPnP1AxisX.alignTablePos.inPos )
      Contact( "Unit1.Em4.ControlNodes".cm.softCam.anodeMainPnP2AxisX.stackTablePos.inPos )
      Coil( "Unit1.Em4.ControlNodes".mainPnP."step".transition1[620] )
   END_RUNG
   RUNG wire#w1
      Contact( "Unit1.Em4.ControlNodes".mainPnP."step".transition1[620] )
      { S7_Templates := "time_type := Time" } #statTonTime[620].TON(pt := #delayTime, et =>)
      Move(in := #JOB_6_STEP_30, out1 => "Unit1.Em4.ControlNodes".mainPnP.sequence.status.nextStep)
   END_RUNG
   // the same network as SCL:
   #_w1 := ("Unit1.Em4.ControlNodes".mainPnP.sequence.status.currentStep = #JOB_6_STEP_20) AND "Unit1.Em4.ControlNodes".mainPnP.sequence.status.seqActive;
   "Unit1.Em4.ControlNodes".mainPnP."step".action1[620] := #_w1 AND (NOT "Unit1.Em4.ControlNodes".cm.softCam.anodeMainPnP1AxisX.alignTablePos.inPos OR NOT "Unit1.Em4.ControlNodes".cm.softCam.anodeMainPnP2AxisX.stackTablePos.inPos);
   "Unit1.Em4.ControlNodes".mainPnP."step".transition1[620] := #_w1 AND "Unit1.Em4.ControlNodes".cm.softCam.anodeMainPnP1AxisX.alignTablePos.inPos AND "Unit1.Em4.ControlNodes".cm.softCam.anodeMainPnP2AxisX.stackTablePos.inPos;
   #statTonTime[620].TON(IN := #_w1 AND "Unit1.Em4.ControlNodes".mainPnP."step".transition1[620],
                         PT := #delayTime);
   IF #statTonTime[620].Q THEN
       "Unit1.Em4.ControlNodes".mainPnP.sequence.status.nextStep := #JOB_6_STEP_30;
   END_IF;
END_REGION

REGION Network 100: Step[630] : Main P&P 1 Rotary Cylinder InWorkPos(=Counter Clock Wise)
   RUNG wire#powerrail
      { S7_Templates := "SrcType := DInt" } EQ_Contact(in1 := "Unit1.Em4.ControlNodes".mainPnP.sequence.status.currentStep, in2 := #JOB_6_STEP_30)
      Contact( "Unit1.Em4.ControlNodes".mainPnP.sequence.status.seqActive )
      wire#w1
      I_Contact( "Unit1.Em4.ControlNodes".cmAnodeMainPnP1RotaryCwCcw.monitoring.inWorkPos )
      Coil( "Unit1.Em4.ControlNodes".mainPnP."step".action1[630] )
   END_RUNG
   RUNG wire#w1
      Contact( "Unit1.Em4.ControlNodes".cmAnodeMainPnP1RotaryCwCcw.monitoring.inWorkPos )
      Coil( "Unit1.Em4.ControlNodes".mainPnP."step".transition1[630] )
   END_RUNG
   RUNG wire#w1
      Contact( "Unit1.Em4.ControlNodes".mainPnP."step".transition1[630] )
      { S7_Templates := "time_type := Time" } #statTonTime[630].TON(pt := #delayTime, et =>)
      Move(in := #JOB_6_STEP_40, out1 => "Unit1.Em4.ControlNodes".mainPnP.sequence.status.nextStep)
   END_RUNG
   // the same network as SCL:
   #_w1 := ("Unit1.Em4.ControlNodes".mainPnP.sequence.status.currentStep = #JOB_6_STEP_30) AND "Unit1.Em4.ControlNodes".mainPnP.sequence.status.seqActive;
   "Unit1.Em4.ControlNodes".mainPnP."step".action1[630] := #_w1 AND NOT "Unit1.Em4.ControlNodes".cmAnodeMainPnP1RotaryCwCcw.monitoring.inWorkPos;
   "Unit1.Em4.ControlNodes".mainPnP."step".transition1[630] := #_w1 AND "Unit1.Em4.ControlNodes".cmAnodeMainPnP1RotaryCwCcw.monitoring.inWorkPos;
   #statTonTime[630].TON(IN := #_w1 AND "Unit1.Em4.ControlNodes".mainPnP."step".transition1[630],
                         PT := #delayTime);
   IF #statTonTime[630].Q THEN
       "Unit1.Em4.ControlNodes".mainPnP.sequence.status.nextStep := #JOB_6_STEP_40;
   END_IF;
END_REGION

REGION Network 101: Step[640] : Main P&P 1 Z-Axis Unload Pos
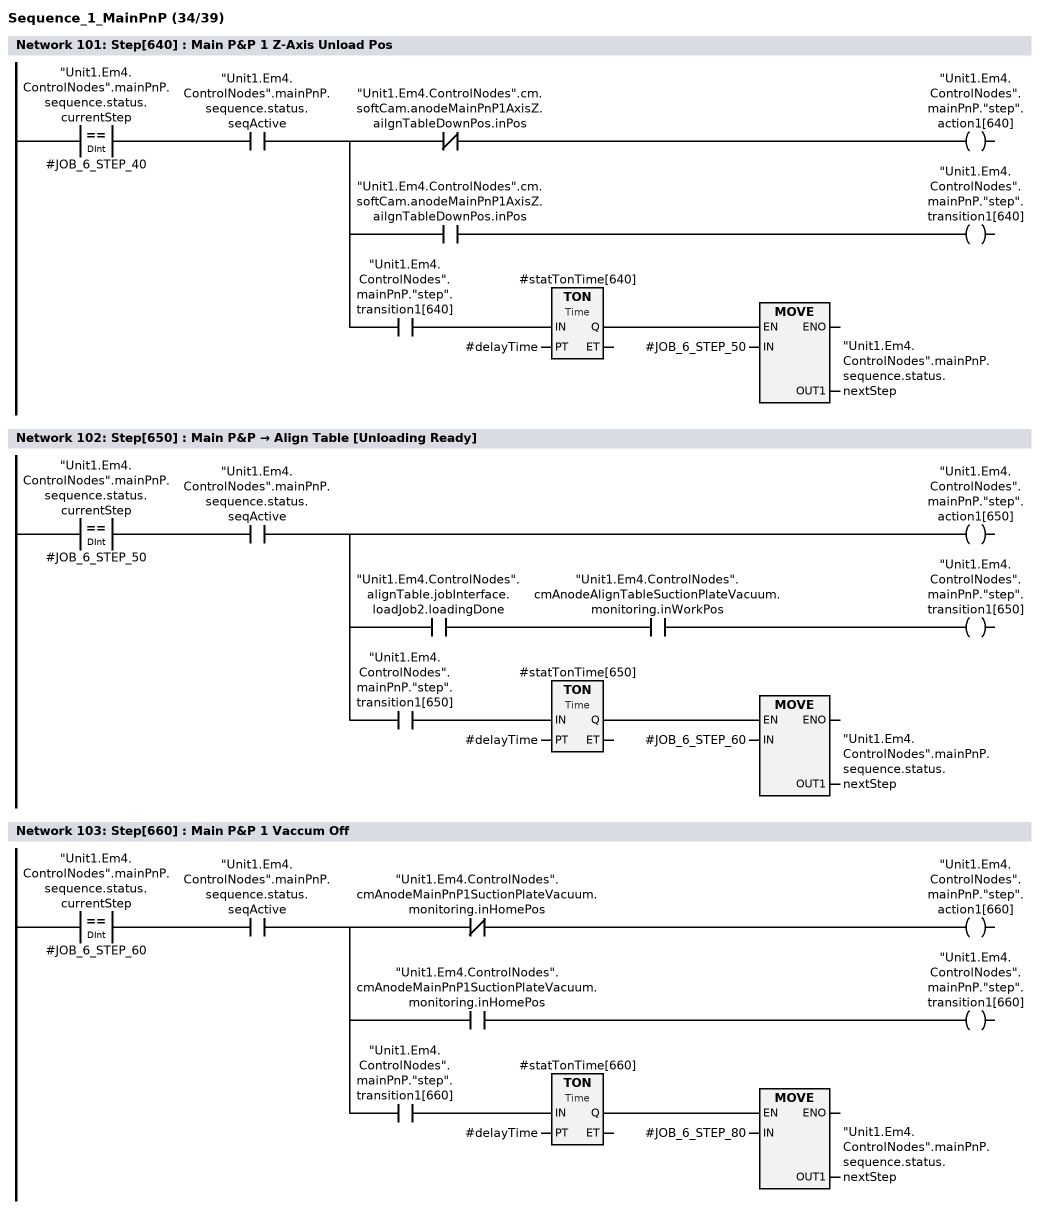
   RUNG wire#powerrail
      { S7_Templates := "SrcType := DInt" } EQ_Contact(in1 := "Unit1.Em4.ControlNodes".mainPnP.sequence.status.currentStep, in2 := #JOB_6_STEP_40)
      Contact( "Unit1.Em4.ControlNodes".mainPnP.sequence.status.seqActive )
      wire#w1
      I_Contact( "Unit1.Em4.ControlNodes".cm.softCam.anodeMainPnP1AxisZ.ailgnTableDownPos.inPos )
      Coil( "Unit1.Em4.ControlNodes".mainPnP."step".action1[640] )
   END_RUNG
   RUNG wire#w1
      Contact( "Unit1.Em4.ControlNodes".cm.softCam.anodeMainPnP1AxisZ.ailgnTableDownPos.inPos )
      Coil( "Unit1.Em4.ControlNodes".mainPnP."step".transition1[640] )
   END_RUNG
   RUNG wire#w1
      Contact( "Unit1.Em4.ControlNodes".mainPnP."step".transition1[640] )
      { S7_Templates := "time_type := Time" } #statTonTime[640].TON(pt := #delayTime, et =>)
      Move(in := #JOB_6_STEP_50, out1 => "Unit1.Em4.ControlNodes".mainPnP.sequence.status.nextStep)
   END_RUNG
   // the same network as SCL:
   #_w1 := ("Unit1.Em4.ControlNodes".mainPnP.sequence.status.currentStep = #JOB_6_STEP_40) AND "Unit1.Em4.ControlNodes".mainPnP.sequence.status.seqActive;
   "Unit1.Em4.ControlNodes".mainPnP."step".action1[640] := #_w1 AND NOT "Unit1.Em4.ControlNodes".cm.softCam.anodeMainPnP1AxisZ.ailgnTableDownPos.inPos;
   "Unit1.Em4.ControlNodes".mainPnP."step".transition1[640] := #_w1 AND "Unit1.Em4.ControlNodes".cm.softCam.anodeMainPnP1AxisZ.ailgnTableDownPos.inPos;
   #statTonTime[640].TON(IN := #_w1 AND "Unit1.Em4.ControlNodes".mainPnP."step".transition1[640],
                         PT := #delayTime);
   IF #statTonTime[640].Q THEN
       "Unit1.Em4.ControlNodes".mainPnP.sequence.status.nextStep := #JOB_6_STEP_50;
   END_IF;
END_REGION

REGION Network 102: Step[650] : Main P&P → Align Table [Unloading Ready]
   RUNG wire#powerrail
      { S7_Templates := "SrcType := DInt" } EQ_Contact(in1 := "Unit1.Em4.ControlNodes".mainPnP.sequence.status.currentStep, in2 := #JOB_6_STEP_50)
      Contact( "Unit1.Em4.ControlNodes".mainPnP.sequence.status.seqActive )
      wire#w1
      Coil( "Unit1.Em4.ControlNodes".mainPnP."step".action1[650] )
   END_RUNG
   RUNG wire#w1
      Contact( "Unit1.Em4.ControlNodes".alignTable.jobInterface.loadJob2.loadingDone )
      Contact( "Unit1.Em4.ControlNodes".cmAnodeAlignTableSuctionPlateVacuum.monitoring.inWorkPos )
      Coil( "Unit1.Em4.ControlNodes".mainPnP."step".transition1[650] )
   END_RUNG
   RUNG wire#w1
      Contact( "Unit1.Em4.ControlNodes".mainPnP."step".transition1[650] )
      { S7_Templates := "time_type := Time" } #statTonTime[650].TON(pt := #delayTime, et =>)
      Move(in := #JOB_6_STEP_60, out1 => "Unit1.Em4.ControlNodes".mainPnP.sequence.status.nextStep)
   END_RUNG
   // the same network as SCL:
   "Unit1.Em4.ControlNodes".mainPnP."step".action1[650] := ("Unit1.Em4.ControlNodes".mainPnP.sequence.status.currentStep = #JOB_6_STEP_50) AND "Unit1.Em4.ControlNodes".mainPnP.sequence.status.seqActive;
   "Unit1.Em4.ControlNodes".mainPnP."step".transition1[650] := ("Unit1.Em4.ControlNodes".mainPnP.sequence.status.currentStep = #JOB_6_STEP_50) AND "Unit1.Em4.ControlNodes".mainPnP.sequence.status.seqActive AND "Unit1.Em4.ControlNodes".alignTable.jobInterface.loadJob2.loadingDone AND "Unit1.Em4.ControlNodes".cmAnodeAlignTableSuctionPlateVacuum.monitoring.inWorkPos;
   #statTonTime[650].TON(IN := ("Unit1.Em4.ControlNodes".mainPnP.sequence.status.currentStep = #JOB_6_STEP_50) AND "Unit1.Em4.ControlNodes".mainPnP.sequence.status.seqActive AND "Unit1.Em4.ControlNodes".mainPnP."step".transition1[650],
                         PT := #delayTime);
   IF #statTonTime[650].Q THEN
       "Unit1.Em4.ControlNodes".mainPnP.sequence.status.nextStep := #JOB_6_STEP_60;
   END_IF;
END_REGION

REGION Network 103: Step[660] : Main P&P 1 Vaccum Off
   RUNG wire#powerrail
      { S7_Templates := "SrcType := DInt" } EQ_Contact(in1 := "Unit1.Em4.ControlNodes".mainPnP.sequence.status.currentStep, in2 := #JOB_6_STEP_60)
      Contact( "Unit1.Em4.ControlNodes".mainPnP.sequence.status.seqActive )
      wire#w1
      I_Contact( "Unit1.Em4.ControlNodes".cmAnodeMainPnP1SuctionPlateVacuum.monitoring.inHomePos )
      Coil( "Unit1.Em4.ControlNodes".mainPnP."step".action1[660] )
   END_RUNG
   RUNG wire#w1
      Contact( "Unit1.Em4.ControlNodes".cmAnodeMainPnP1SuctionPlateVacuum.monitoring.inHomePos )
      Coil( "Unit1.Em4.ControlNodes".mainPnP."step".transition1[660] )
   END_RUNG
   RUNG wire#w1
      Contact( "Unit1.Em4.ControlNodes".mainPnP."step".transition1[660] )
      { S7_Templates := "time_type := Time" } #statTonTime[660].TON(pt := #delayTime, et =>)
      Move(in := #JOB_6_STEP_80, out1 => "Unit1.Em4.ControlNodes".mainPnP.sequence.status.nextStep)
   END_RUNG
   // the same network as SCL:
   #_w1 := ("Unit1.Em4.ControlNodes".mainPnP.sequence.status.currentStep = #JOB_6_STEP_60) AND "Unit1.Em4.ControlNodes".mainPnP.sequence.status.seqActive;
   "Unit1.Em4.ControlNodes".mainPnP."step".action1[660] := #_w1 AND NOT "Unit1.Em4.ControlNodes".cmAnodeMainPnP1SuctionPlateVacuum.monitoring.inHomePos;
   "Unit1.Em4.ControlNodes".mainPnP."step".transition1[660] := #_w1 AND "Unit1.Em4.ControlNodes".cmAnodeMainPnP1SuctionPlateVacuum.monitoring.inHomePos;
   #statTonTime[660].TON(IN := #_w1 AND "Unit1.Em4.ControlNodes".mainPnP."step".transition1[660],
                         PT := #delayTime);
   IF #statTonTime[660].Q THEN
       "Unit1.Em4.ControlNodes".mainPnP.sequence.status.nextStep := #JOB_6_STEP_80;
   END_IF;
END_REGION

REGION Network 104: Step[680] : Main P&P 1 Z-Axis Wait Pos
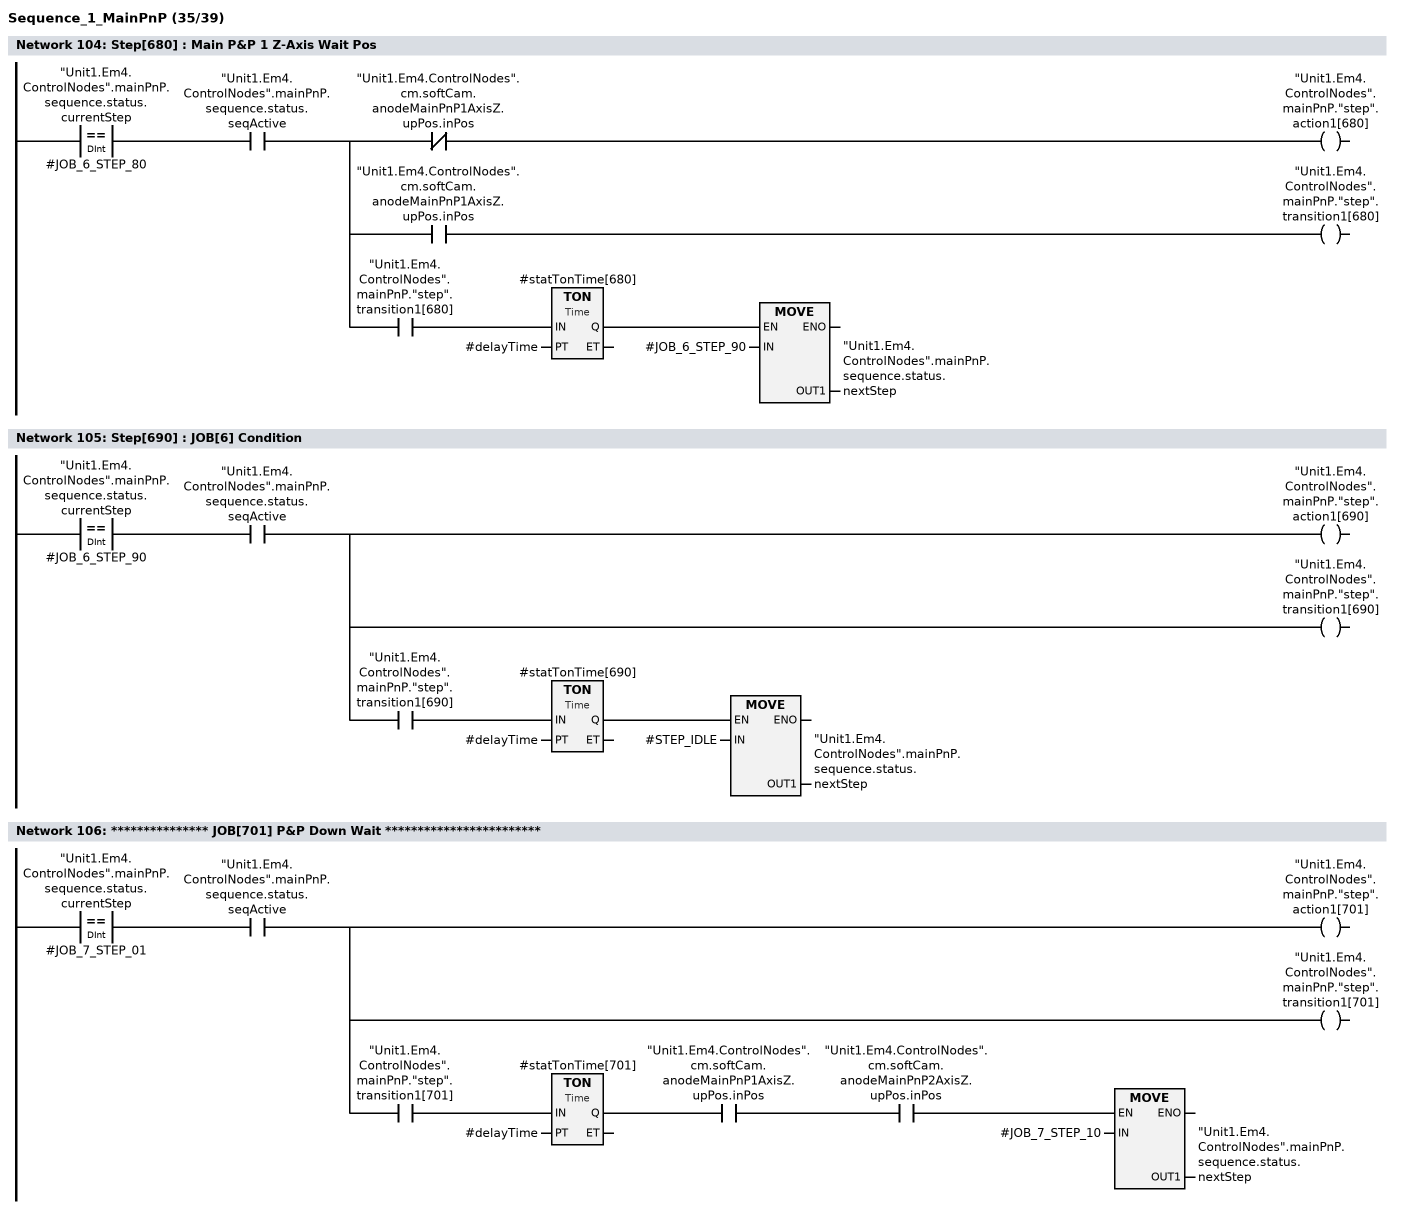
   RUNG wire#powerrail
      { S7_Templates := "SrcType := DInt" } EQ_Contact(in1 := "Unit1.Em4.ControlNodes".mainPnP.sequence.status.currentStep, in2 := #JOB_6_STEP_80)
      Contact( "Unit1.Em4.ControlNodes".mainPnP.sequence.status.seqActive )
      wire#w1
      I_Contact( "Unit1.Em4.ControlNodes".cm.softCam.anodeMainPnP1AxisZ.upPos.inPos )
      Coil( "Unit1.Em4.ControlNodes".mainPnP."step".action1[680] )
   END_RUNG
   RUNG wire#w1
      Contact( "Unit1.Em4.ControlNodes".cm.softCam.anodeMainPnP1AxisZ.upPos.inPos )
      Coil( "Unit1.Em4.ControlNodes".mainPnP."step".transition1[680] )
   END_RUNG
   RUNG wire#w1
      Contact( "Unit1.Em4.ControlNodes".mainPnP."step".transition1[680] )
      { S7_Templates := "time_type := Time" } #statTonTime[680].TON(pt := #delayTime, et =>)
      Move(in := #JOB_6_STEP_90, out1 => "Unit1.Em4.ControlNodes".mainPnP.sequence.status.nextStep)
   END_RUNG
   // the same network as SCL:
   #_w1 := ("Unit1.Em4.ControlNodes".mainPnP.sequence.status.currentStep = #JOB_6_STEP_80) AND "Unit1.Em4.ControlNodes".mainPnP.sequence.status.seqActive;
   "Unit1.Em4.ControlNodes".mainPnP."step".action1[680] := #_w1 AND NOT "Unit1.Em4.ControlNodes".cm.softCam.anodeMainPnP1AxisZ.upPos.inPos;
   "Unit1.Em4.ControlNodes".mainPnP."step".transition1[680] := #_w1 AND "Unit1.Em4.ControlNodes".cm.softCam.anodeMainPnP1AxisZ.upPos.inPos;
   #statTonTime[680].TON(IN := #_w1 AND "Unit1.Em4.ControlNodes".mainPnP."step".transition1[680],
                         PT := #delayTime);
   IF #statTonTime[680].Q THEN
       "Unit1.Em4.ControlNodes".mainPnP.sequence.status.nextStep := #JOB_6_STEP_90;
   END_IF;
END_REGION

REGION Network 105: Step[690] : JOB[6] Condition
   RUNG wire#powerrail
      { S7_Templates := "SrcType := DInt" } EQ_Contact(in1 := "Unit1.Em4.ControlNodes".mainPnP.sequence.status.currentStep, in2 := #JOB_6_STEP_90)
      Contact( "Unit1.Em4.ControlNodes".mainPnP.sequence.status.seqActive )
      wire#w1
      Coil( "Unit1.Em4.ControlNodes".mainPnP."step".action1[690] )
   END_RUNG
   RUNG wire#w1
      Coil( "Unit1.Em4.ControlNodes".mainPnP."step".transition1[690] )
   END_RUNG
   RUNG wire#w1
      Contact( "Unit1.Em4.ControlNodes".mainPnP."step".transition1[690] )
      { S7_Templates := "time_type := Time" } #statTonTime[690].TON(pt := #delayTime, et =>)
      Move(in := #STEP_IDLE, out1 => "Unit1.Em4.ControlNodes".mainPnP.sequence.status.nextStep)
   END_RUNG
   // the same network as SCL:
   "Unit1.Em4.ControlNodes".mainPnP."step".action1[690] := ("Unit1.Em4.ControlNodes".mainPnP.sequence.status.currentStep = #JOB_6_STEP_90) AND "Unit1.Em4.ControlNodes".mainPnP.sequence.status.seqActive;
   "Unit1.Em4.ControlNodes".mainPnP."step".transition1[690] := ("Unit1.Em4.ControlNodes".mainPnP.sequence.status.currentStep = #JOB_6_STEP_90) AND "Unit1.Em4.ControlNodes".mainPnP.sequence.status.seqActive;
   #statTonTime[690].TON(IN := ("Unit1.Em4.ControlNodes".mainPnP.sequence.status.currentStep = #JOB_6_STEP_90) AND "Unit1.Em4.ControlNodes".mainPnP.sequence.status.seqActive AND "Unit1.Em4.ControlNodes".mainPnP."step".transition1[690],
                         PT := #delayTime);
   IF #statTonTime[690].Q THEN
       "Unit1.Em4.ControlNodes".mainPnP.sequence.status.nextStep := #STEP_IDLE;
   END_IF;
END_REGION

REGION Network 106: *************** JOB[701] P&P Down Wait ************************
   RUNG wire#powerrail
      { S7_Templates := "SrcType := DInt" } EQ_Contact(in1 := "Unit1.Em4.ControlNodes".mainPnP.sequence.status.currentStep, in2 := #JOB_7_STEP_01)
      Contact( "Unit1.Em4.ControlNodes".mainPnP.sequence.status.seqActive )
      wire#w1
      Coil( "Unit1.Em4.ControlNodes".mainPnP."step".action1[701] )
   END_RUNG
   RUNG wire#w1
      Coil( "Unit1.Em4.ControlNodes".mainPnP."step".transition1[701] )
   END_RUNG
   RUNG wire#w1
      Contact( "Unit1.Em4.ControlNodes".mainPnP."step".transition1[701] )
      { S7_Templates := "time_type := Time" } #statTonTime[701].TON(pt := #delayTime, et =>)
      Contact( "Unit1.Em4.ControlNodes".cm.softCam.anodeMainPnP1AxisZ.upPos.inPos )
      Contact( "Unit1.Em4.ControlNodes".cm.softCam.anodeMainPnP2AxisZ.upPos.inPos )
      Move(in := #JOB_7_STEP_10, out1 => "Unit1.Em4.ControlNodes".mainPnP.sequence.status.nextStep)
   END_RUNG
   // the same network as SCL:
   "Unit1.Em4.ControlNodes".mainPnP."step".action1[701] := ("Unit1.Em4.ControlNodes".mainPnP.sequence.status.currentStep = #JOB_7_STEP_01) AND "Unit1.Em4.ControlNodes".mainPnP.sequence.status.seqActive;
   "Unit1.Em4.ControlNodes".mainPnP."step".transition1[701] := ("Unit1.Em4.ControlNodes".mainPnP.sequence.status.currentStep = #JOB_7_STEP_01) AND "Unit1.Em4.ControlNodes".mainPnP.sequence.status.seqActive;
   #statTonTime[701].TON(IN := ("Unit1.Em4.ControlNodes".mainPnP.sequence.status.currentStep = #JOB_7_STEP_01) AND "Unit1.Em4.ControlNodes".mainPnP.sequence.status.seqActive AND "Unit1.Em4.ControlNodes".mainPnP."step".transition1[701],
                         PT := #delayTime);
   IF #statTonTime[701].Q AND "Unit1.Em4.ControlNodes".cm.softCam.anodeMainPnP1AxisZ.upPos.inPos AND "Unit1.Em4.ControlNodes".cm.softCam.anodeMainPnP2AxisZ.upPos.inPos THEN
       "Unit1.Em4.ControlNodes".mainPnP.sequence.status.nextStep := #JOB_7_STEP_10;
   END_IF;
END_REGION

REGION Network 107: Step[710] : Z1,z2 axis up pos move
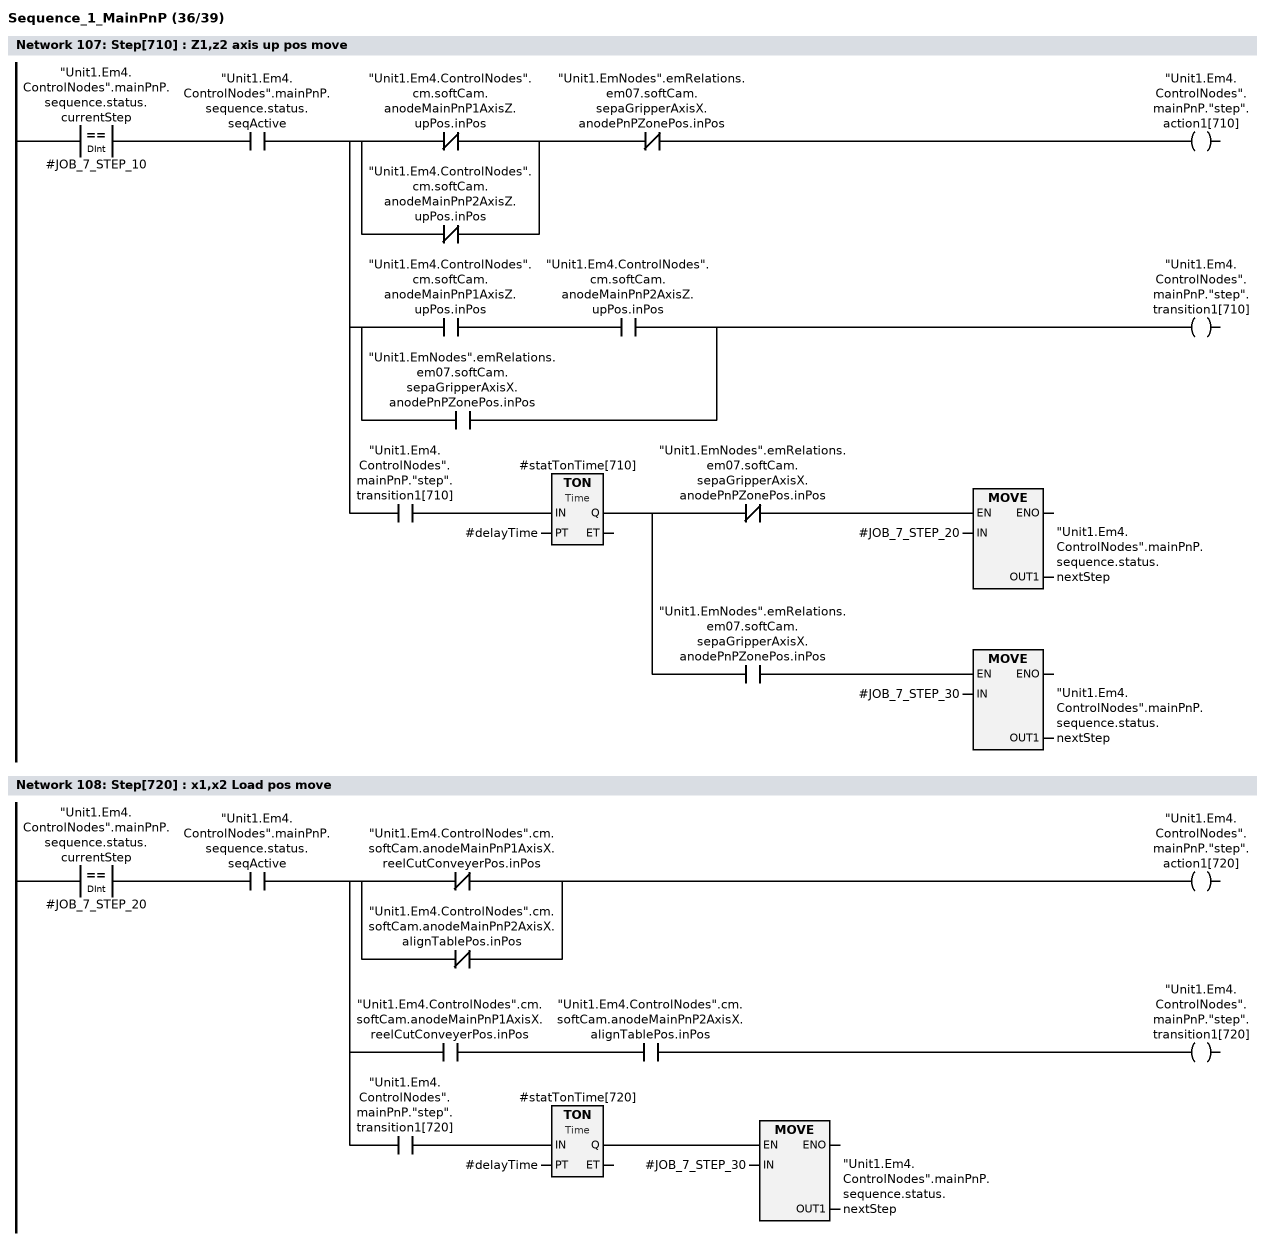
   RUNG wire#powerrail
      { S7_Templates := "SrcType := DInt" } EQ_Contact(in1 := "Unit1.Em4.ControlNodes".mainPnP.sequence.status.currentStep, in2 := #JOB_7_STEP_10)
      Contact( "Unit1.Em4.ControlNodes".mainPnP.sequence.status.seqActive )
      wire#w1
      I_Contact( "Unit1.Em4.ControlNodes".cm.softCam.anodeMainPnP1AxisZ.upPos.inPos )
      wire#w2
      I_Contact( "Unit1.EmNodes".emRelations.em07.softCam.sepaGripperAxisX.anodePnPZonePos.inPos )
      Coil( "Unit1.Em4.ControlNodes".mainPnP."step".action1[710] )
   END_RUNG
   RUNG wire#w1
      I_Contact( "Unit1.Em4.ControlNodes".cm.softCam.anodeMainPnP2AxisZ.upPos.inPos )
   END_RUNG wire#w2
   RUNG wire#w1
      Contact( "Unit1.Em4.ControlNodes".cm.softCam.anodeMainPnP1AxisZ.upPos.inPos )
      Contact( "Unit1.Em4.ControlNodes".cm.softCam.anodeMainPnP2AxisZ.upPos.inPos )
      wire#w3
      Coil( "Unit1.Em4.ControlNodes".mainPnP."step".transition1[710] )
   END_RUNG
   RUNG wire#w1
      Contact( "Unit1.EmNodes".emRelations.em07.softCam.sepaGripperAxisX.anodePnPZonePos.inPos )
   END_RUNG wire#w3
   RUNG wire#w1
      Contact( "Unit1.Em4.ControlNodes".mainPnP."step".transition1[710] )
      { S7_Templates := "time_type := Time" } #statTonTime[710].TON(pt := #delayTime, et =>)
      wire#w4
      I_Contact( "Unit1.EmNodes".emRelations.em07.softCam.sepaGripperAxisX.anodePnPZonePos.inPos )
      Move(in := #JOB_7_STEP_20, out1 => "Unit1.Em4.ControlNodes".mainPnP.sequence.status.nextStep)
   END_RUNG
   RUNG wire#w4
      Contact( "Unit1.EmNodes".emRelations.em07.softCam.sepaGripperAxisX.anodePnPZonePos.inPos )
      Move(in := #JOB_7_STEP_30, out1 => "Unit1.Em4.ControlNodes".mainPnP.sequence.status.nextStep)
   END_RUNG
   // the same network as SCL:
   #_w1 := ("Unit1.Em4.ControlNodes".mainPnP.sequence.status.currentStep = #JOB_7_STEP_10) AND "Unit1.Em4.ControlNodes".mainPnP.sequence.status.seqActive;
   "Unit1.Em4.ControlNodes".mainPnP."step".action1[710] := #_w1 AND (NOT "Unit1.Em4.ControlNodes".cm.softCam.anodeMainPnP1AxisZ.upPos.inPos OR NOT "Unit1.Em4.ControlNodes".cm.softCam.anodeMainPnP2AxisZ.upPos.inPos) AND NOT "Unit1.EmNodes".emRelations.em07.softCam.sepaGripperAxisX.anodePnPZonePos.inPos;
   "Unit1.Em4.ControlNodes".mainPnP."step".transition1[710] := #_w1 AND (("Unit1.Em4.ControlNodes".cm.softCam.anodeMainPnP1AxisZ.upPos.inPos AND "Unit1.Em4.ControlNodes".cm.softCam.anodeMainPnP2AxisZ.upPos.inPos) OR "Unit1.EmNodes".emRelations.em07.softCam.sepaGripperAxisX.anodePnPZonePos.inPos);
   #statTonTime[710].TON(IN := #_w1 AND "Unit1.Em4.ControlNodes".mainPnP."step".transition1[710],
                         PT := #delayTime);
   IF #statTonTime[710].Q AND NOT "Unit1.EmNodes".emRelations.em07.softCam.sepaGripperAxisX.anodePnPZonePos.inPos THEN
       "Unit1.Em4.ControlNodes".mainPnP.sequence.status.nextStep := #JOB_7_STEP_20;
   END_IF;
   IF #statTonTime[710].Q AND "Unit1.EmNodes".emRelations.em07.softCam.sepaGripperAxisX.anodePnPZonePos.inPos THEN
       "Unit1.Em4.ControlNodes".mainPnP.sequence.status.nextStep := #JOB_7_STEP_30;
   END_IF;
END_REGION

REGION Network 108: Step[720] : x1,x2 Load pos move
   RUNG wire#powerrail
      { S7_Templates := "SrcType := DInt" } EQ_Contact(in1 := "Unit1.Em4.ControlNodes".mainPnP.sequence.status.currentStep, in2 := #JOB_7_STEP_20)
      Contact( "Unit1.Em4.ControlNodes".mainPnP.sequence.status.seqActive )
      wire#w1
      I_Contact( "Unit1.Em4.ControlNodes".cm.softCam.anodeMainPnP1AxisX.reelCutConveyerPos.inPos )
      wire#w2
      Coil( "Unit1.Em4.ControlNodes".mainPnP."step".action1[720] )
   END_RUNG
   RUNG wire#w1
      I_Contact( "Unit1.Em4.ControlNodes".cm.softCam.anodeMainPnP2AxisX.alignTablePos.inPos )
   END_RUNG wire#w2
   RUNG wire#w1
      Contact( "Unit1.Em4.ControlNodes".cm.softCam.anodeMainPnP1AxisX.reelCutConveyerPos.inPos )
      Contact( "Unit1.Em4.ControlNodes".cm.softCam.anodeMainPnP2AxisX.alignTablePos.inPos )
      Coil( "Unit1.Em4.ControlNodes".mainPnP."step".transition1[720] )
   END_RUNG
   RUNG wire#w1
      Contact( "Unit1.Em4.ControlNodes".mainPnP."step".transition1[720] )
      { S7_Templates := "time_type := Time" } #statTonTime[720].TON(pt := #delayTime, et =>)
      Move(in := #JOB_7_STEP_30, out1 => "Unit1.Em4.ControlNodes".mainPnP.sequence.status.nextStep)
   END_RUNG
   // the same network as SCL:
   #_w1 := ("Unit1.Em4.ControlNodes".mainPnP.sequence.status.currentStep = #JOB_7_STEP_20) AND "Unit1.Em4.ControlNodes".mainPnP.sequence.status.seqActive;
   "Unit1.Em4.ControlNodes".mainPnP."step".action1[720] := #_w1 AND (NOT "Unit1.Em4.ControlNodes".cm.softCam.anodeMainPnP1AxisX.reelCutConveyerPos.inPos OR NOT "Unit1.Em4.ControlNodes".cm.softCam.anodeMainPnP2AxisX.alignTablePos.inPos);
   "Unit1.Em4.ControlNodes".mainPnP."step".transition1[720] := #_w1 AND "Unit1.Em4.ControlNodes".cm.softCam.anodeMainPnP1AxisX.reelCutConveyerPos.inPos AND "Unit1.Em4.ControlNodes".cm.softCam.anodeMainPnP2AxisX.alignTablePos.inPos;
   #statTonTime[720].TON(IN := #_w1 AND "Unit1.Em4.ControlNodes".mainPnP."step".transition1[720],
                         PT := #delayTime);
   IF #statTonTime[720].Q THEN
       "Unit1.Em4.ControlNodes".mainPnP.sequence.status.nextStep := #JOB_7_STEP_30;
   END_IF;
END_REGION

